(*								ELSIF iVisionScanModel=0 THEN
									(* found nothing, check if there is a part *)
									IF bRetryVision THEN
										sCurrentState.eStep := SP_RunStp103;
										bRetryVision := FALSE;
									ELSE
										sCurrentState.eStep := SP_RunStp120;
									END_IF
								ELSIF iVisionScanModel < iMaxScanVisionModelPart THEN
									(* relaunch scan with next step model *)
									iVisionScanModel := iVisionScanModel + 1;
									sCurrentState.eStep := SP_RunStp105;
								ELSE
									(* Part cannot be recognize, skip to next one *)
									aTPartOnPlate[LPP_Lift1,iPlatePos].ePartStatus := PPS_BadPart;
									iPlatePos := iPlatePos + 1;
									sCurrentState.eStep := SP_RunStp102;
*)								END_IF
							END_IF
						SP_RunStp110: (* Found valid position, Get Z position *)
							IF bUse103171OptimB3 THEN
								IF (alrZLiftPos[LTP_Lift1] = 0) THEN
									eScanPos := LTP_Lift1;
									eReturnStepMeasureZLift := SP_RunStp110;
									sCurrentState.eStep := SP_RunStp500;
								ELSE
									ZPositionTakeGive := alrRobotPos[LTA_Z,LTP_TableSideALayering1] + alrRobotOffset[LTA_Z, iHead] + (lrCalibrationPartAndHeadHeight - sPartDataMMI.lrPartAndHeadHeight) - alrZLiftPos[LTP_Lift1] - lrZSensorCalibrationOffset;
									sCurrentState.eStep := SP_RunStp114;
								END_IF
							ELSE
								iZSensorPositionScan := 0;
								sCurrentState.eStep := SP_RunStp111;
							END_IF
						SP_RunStp111:
							alrSecuredTarget[LA_X] := alrRobotPos[LTA_X,LTP_Lift1] + alrRobotOffset[LTA_X, LTO_ZSensor] + alrLiftCalibrationOffset[LTP_Lift1,LTA_X]  -  sPlateData.alrPartOnPlate[iPlatePos].lrX - sPartDataMMI.alrSensorZOffset[iZSensorPositionScan].lrX;
							alrSecuredTarget[LA_Y] :=alrRobotPos[LTA_Y,LTP_Lift1] + alrRobotOffset[LTA_Y, LTO_ZSensor] + alrLiftCalibrationOffset[LTP_Lift1,LTA_Y] - sPlateData.alrPartOnPlate[iPlatePos].lrY - sPartDataMMI.alrSensorZOffset[iZSensorPositionScan].lrY;
							TSensorZWaitStab(IN := FALSE);
							sCurrentState.bWaitStep := TRUE;
							eReturnStep4SecureMove := SP_RunStp112;
							sCurrentState.eStep := SP_RunStp550;
						SP_RunStp112:
							IF eRobotXYTStatus = AS_InPosition THEN
								TSensorZWaitStab(IN := TRUE, PT := TSensorZWaitStabTime);
								IF TSensorZWaitStab.Q THEN
									IF TSensorMeasure.bInputOutOfRange THEN
										bZSensorOutOfRangeError := TRUE;
									END_IF
									lrZSensorPosition[iZSensorPositionScan] := TSensorMeasure.lrValue;
									IF iZSensorPositionScan = 0 AND (sPartDataMMI.alrSensorZOffset[1].lrX<>0 OR sPartDataMMI.alrSensorZOffset[1].lrY<>0) THEN
										iZSensorPositionScan := iZSensorPositionScan + 1;
										sCurrentState.eStep := SP_RunStp111;
									ELSE
										sCurrentState.eStep := SP_RunStp113;
									END_IF
								END_IF
							END_IF
						SP_RunStp113:
							IF iZSensorPositionScan = 1 THEN
								(* We used two position, mean the value *)
								ZPositionTakeGive := (lrZSensorPosition[0] + lrZSensorPosition[1]) / 2;
							ELSE
								(* Only one position, use the first one then *)
								ZPositionTakeGive := lrZSensorPosition[0];
							END_IF
							ZPositionTakeGive := alrRobotPos[LTA_Z,LTP_TableSideALayering1] + alrRobotOffset[LTA_Z, iHead] + (lrCalibrationPartAndHeadHeight - sPartDataMMI.lrPartAndHeadHeight) - ZPositionTakeGive;
							sCurrentState.eStep := SP_RunStp114;
						SP_RunStp114: (* Move to take position *)
							IF sRunDataVision.TVisionPartData.bPresent AND NOT sRunDataVision.TVisionPartData.bValid THEN
								alrSecuredTarget[LA_X] := alrRobotPos[LTA_X,LTP_Lift1] + alrRobotOffset[LTA_X, iHead] + alrLiftCalibrationOffset[LTP_Lift1,LTA_X]  -  sPlateData.alrPartOnPlate[iPlatePos].lrX;	// + INT(iPlatePos/5) * 1/9 * offsetXMax;		// HFO : when vision diseable, correct the offset X between parts 
								alrSecuredTarget[LA_Y] :=alrRobotPos[LTA_Y,LTP_Lift1] + alrRobotOffset[LTA_Y, iHead] + alrLiftCalibrationOffset[LTP_Lift1,LTA_Y] - sPlateData.alrPartOnPlate[iPlatePos].lrY;	// + int(iPlatePos%5) * 1/4 * offsetYMax;		// HFO : when vision diseable, correct the offset Y between parts 
								alrTargetPos[LA_THETA] := alrRobotPos[LTA_THETA,LTP_TableSideALayering1] + alrRobotOffset[LTA_THETA, iHead] - (-90);
							ELSE
								alrSecuredTarget[LA_X] := alrRobotPos[LTA_X,LTP_Lift1] + alrRobotOffset[LTA_X, iHead] + alrLiftCalibrationOffset[LTP_Lift1,LTA_X]  -  sPlateData.alrPartOnPlate[iPlatePos].lrX + sRunDataVision.TVisionPartData.lrX;
								alrSecuredTarget[LA_Y] :=alrRobotPos[LTA_Y,LTP_Lift1] + alrRobotOffset[LTA_Y, iHead] + alrLiftCalibrationOffset[LTP_Lift1,LTA_Y] - sPlateData.alrPartOnPlate[iPlatePos].lrY + sRunDataVision.TVisionPartData.lrY;
								alrTargetPos[LA_THETA] := alrRobotPos[LTA_THETA,LTP_TableSideALayering1] + alrRobotOffset[LTA_THETA, iHead] + (360 - sRunDataVision.TVisionPartData.lrTheta);
							END_IF
							aeMoveRobotCommand[LA_THETA] := AC_MoveAtAbsPos;
							eReturnStep4SecureMove := SP_RunStp115;
							sCurrentState.eStep := SP_RunStp550;
						SP_RunStp115:
							IF eRobotXYTStatus = AS_InPosition THEN
								sCurrentState.eStep := SP_RunStp1;
							END_IF
						SP_RunStp120: (*Scan Vision Empty position *)
							sRunDataVision.iUseModel := iVisionModelEmpty;
							eVisionRunCmd := RCV_AnalyseImage;
							sCurrentState.eStep := SP_RunStp121;
						SP_RunStp121: (* Check for empty position *)
							IF eVisionRunStatus = RS_WaitRequest THEN
								IF NOT sRunDataVision.TVisionPartData.bPresent THEN
									(* Found Empty Position *)
									aTPartOnPlate[LPP_Lift1,iPlatePos].ePartStatus := PPS_Absent;
									iPlatePos := iPlatePos + 1;
									sCurrentState.eStep := SP_RunStp102;
								ELSE
									(*  Position is not empty, part is not recognize*)
									iVisionScanModel := iVisionScanModel + 1;
									sCurrentState.eStep := SP_RunStp104;
								END_IF
							END_IF
						SP_RunStp150: (* Switch plate *)
							bInvalidPlate := FALSE;
							FOR iPlatePos := 0 TO sPlateData.iNbPartOnPlate-1 DO
								IF aTPartOnPlate[LPP_Lift1,iPlatePos].ePartStatus = PPS_BadPart THEN
//									bInvalidPlate := TRUE;
									EXIT;
								END_IF
							END_FOR
							IF bInvalidPlate THEN
								(* goto invalid plate *)
								bLift1Lift1BadPlate := TRUE;
								eLift1RunCmd := RCL_MoveToOpenDrawer;
								sCurrentState.eStep := SP_RunStp101;
							ELSE
								sCurrentState.eStep := SP_RunStp70; (* Call Switch Plate *)
								eReturnStep := SP_RunStp101;
							END_IF
						SP_RunStp170: (*Get from Table *)
							IF eTableSide = TS_A THEN
								IF sRunData.iLayringPos = 0 THEN
									ePos := LTP_TableSideALayering1;
								ELSE
									ePos := LTP_TableSideALayering2;
								END_IF
							ELSE
								IF sRunData.iLayringPos = 0 THEN
									ePos := LTP_TableSideBLayering1;
								ELSE
									ePos := LTP_TableSideBLayering2;
								END_IF
							END_IF
							alrSecuredTarget[LA_X] := alrRobotPos[LTA_X,ePos] + alrRobotOffset[LTA_X, iHead];
							alrSecuredTarget[LA_Y] :=  alrRobotPos[LTA_Y,ePos] + alrRobotOffset[LTA_Y, iHead];
							alrTargetPos[LA_THETA] := alrRobotPos[LTA_THETA,ePos] + alrRobotOffset[LTA_THETA, iHead];
							ZPositionTakeGive := alrRobotPos[LTA_Z,ePos] + alrRobotOffset[LTA_Z, iHead];
							alrSecuredTarget[LA_X] := alrSecuredTarget[LA_X]   -  sPartDataMMI.alrPartOffsetLayering[sRunData.iLayringOffsetPos].lrX;
							alrSecuredTarget[LA_Y] := alrSecuredTarget[LA_Y]  + sPartDataMMI.alrPartOffsetLayering[sRunData.iLayringOffsetPos].lrY;
							ZPositionTakeGive := ZPositionTakeGive + (lrCalibrationLayeringAndPartAndHeadHeight - sPartDataMMI.lrLayeringAndPartAndHeadHeight);
							aeMoveRobotCommand[LA_THETA] := AC_MoveAtAbsPos;
							eReturnStep4SecureMove := SP_RunStp171;
							sCurrentState.eStep := SP_RunStp550;
						SP_RunStp171:
							IF eRobotXYTStatus = AS_InPosition THEN
								sCurrentState.eStep := SP_RunStp1;
							END_IF
						SP_RunStp180: (*Get from Turn Over *)
							alrSecuredTarget[LA_X] := alrRobotPos[LTA_X,LTP_TurnOverFix] + alrRobotOffset[LTA_X, iHead];
							alrSecuredTarget[LA_Y] :=  alrRobotPos[LTA_Y,LTP_TurnOverFix] + alrRobotOffset[LTA_Y, iHead];
							alrTargetPos[LA_THETA] := alrRobotPos[LTA_THETA,LTP_TurnOverFix] + alrRobotOffset[LTA_THETA, iHead];
							ZPositionTakeGive := alrRobotPos[LTA_Z,LTP_TurnOverFix] + alrRobotOffset[LTA_Z, iHead];
							ZPositionTakeGive := ZPositionTakeGive +  (lrCalibrationLayeringAndPartAndHeadHeight - sPartDataMMI.lrLayeringAndPartAndHeadHeight);
							aeMoveRobotCommand[LA_THETA] := AC_MoveAtAbsPos;
							eReturnStep4SecureMove := SP_RunStp181;
							sCurrentState.eStep := SP_RunStp550;
						SP_RunStp181:
							IF eRobotXYTStatus = AS_InPosition THEN
								sCurrentState.eStep := SP_RunStp1;
							END_IF
						SP_RunStp200 : (*Prepare for Drop part*)
							CASE sRunData.eModule OF
								LMP_Reject, LMP_Sample:
									sCurrentState.eStep := SP_RunStp301;
								LMP_Lift2:
									IF sPartDataMMI.bDropInBox THEN
										sCurrentState.eStep := SP_RunStp230;
									ELSE
										sCurrentState.eStep := SP_RunStp201;
									END_IF
								LMP_Table:
									sCurrentState.eStep := SP_RunStp270;
								LMP_TurnOverArm:
									sCurrentState.eStep := SP_RunStp280;
							END_CASE
						SP_RunStp201: (* Check Lift Status*)
							IF eLift2RunStatus = RS_WaitRequest THEN
								CASE sLift2RunData.eLiftPos OF
									LP_OnPlate:
										iPlatePos := 0;
										sCurrentState.eStep := SP_RunStp202;
									LP_Full,LP_Empty:
										bLift2NeedsPlate := TRUE;
										eLift2RunCmd := RCL_MoveToOpenDrawer;
								ELSE
									eLift2RunCmd := RCL_MoveToPlate;
								END_CASE
							END_IF
						SP_RunStp202: (*Check part status*)
							bFoundPlatePos := FALSE;
							WHILE (iPlatePos < sPlateData.iNbPartOnPlate) DO
								IF aTPartOnPlate[LPP_Lift2,iPlatePos].ePartStatus = PPS_Absent OR aTPartOnPlate[LPP_Lift2,iPlatePos].ePartStatus = PPS_Undefined THEN
									bFoundPlatePos := TRUE;
									EXIT;
								ELSE
									iPlatePos := iPlatePos + 1;
								END_IF
							END_WHILE
							IF NOT bFoundPlatePos THEN
								(* Goto switch plate *)
								sCurrentState.eStep := SP_RunStp250;
							ELSE
								IF aTPartOnPlate[LPP_Lift2,iPlatePos].ePartStatus = PPS_Absent OR (NOT sPlateData.bUseVisionForDrop OR bDisableVision) THEN
									sCurrentState.eStep := SP_RunStp210;
								ELSE
									sCurrentState.eStep := SP_RunStp203;
								END_IF
							END_IF
						SP_RunStp203: (*Scan Vision Part Position *)
							alrSecuredTarget[LA_X] := alrRobotPos[LTA_X,LTP_Lift2] + alrRobotOffset[LTA_X, LTO_Vision] + alrLiftCalibrationOffset[LTP_Lift2,LTA_X]  - sPlateData.alrPartOnPlate[iPlatePos].lrX ;
							alrSecuredTarget[LA_Y] :=  alrRobotPos[LTA_Y,LTP_Lift2] + alrRobotOffset[LTA_Y, LTO_Vision] + alrLiftCalibrationOffset[LTP_Lift2,LTA_Y] - sPlateData.alrPartOnPlate[iPlatePos].lrY ;
							iVisionScanModel := 0;
							TVisionWaitStab(IN := FALSE);
							eReturnStep4SecureMove := SP_RunStp204;
							sCurrentState.eStep := SP_RunStp550;
						SP_RunStp204:
							IF eRobotXYTStatus = AS_InPosition THEN
								IF aTPartOnPlate[LPP_Lift2,iPlatePos].ePartStatus = PPS_Absent THEN
									sCurrentState.eStep := SP_RunStp208;
								ELSE
									TVisionWaitStab(IN := TRUE, PT := TVisionWaitStabTime);
									IF TVisionWaitStab.Q THEN
										eVisionRunCmd := RCV_GrabImage;
										sCurrentState.eStep := SP_RunStp205;
									END_IF
								END_IF
							END_IF
						SP_RunStp205: (* Move to pre-drop position *)
							IF eVisionRunStatus = RS_WaitRequest THEN
								IF bUse103171OptimB5PreMoveXY THEN
									alrSecuredTarget[LA_X] := alrRobotPos[LTA_X,LTP_Lift2] + alrRobotOffset[LTA_X, iHead] + alrLiftCalibrationOffset[LTP_Lift2,LTA_X]  -  sPlateData.alrPartOnPlate[iPlatePos].lrX;
									alrSecuredTarget[LA_Y] :=alrRobotPos[LTA_Y,LTP_Lift2] + alrRobotOffset[LTA_Y, iHead] + alrLiftCalibrationOffset[LTP_Lift2,LTA_Y] - sPlateData.alrPartOnPlate[iPlatePos].lrY;
									alrTargetPos[LA_THETA] := alrRobotPos[LTA_THETA,LTP_TableSideALayering1] + alrRobotOffset[LTA_THETA, iHead];
									aeMoveRobotCommand[LA_THETA] := AC_MoveAtAbsPos;
									eReturnStep4SecureMove := SP_RunStp207;
									sCurrentState.eStep := SP_RunStp550;
								ELSE
									sCurrentState.eStep := SP_RunStp207;
								END_IF
								sRunDataVision.iUseModel := iVisionModelEmpty;
								eVisionRunCmd := RCV_AnalyseImage;
							END_IF
						SP_RunStp207: (* Check for part *)
							IF eVisionRunStatus = RS_WaitRequest THEN
								IF NOT sRunDataVision.TVisionPartData.bPresent THEN
									(* Found empty position *)
									aTPartOnPlate[LPP_Lift2,iPlatePos].ePartStatus := PPS_Absent;
									sCurrentState.eStep := SP_RunStp208;
								ELSE
									(* found something *)
									aTPartOnPlate[LPP_Lift2,iPlatePos].ePartStatus := PPS_Present;
									iPlatePos := iPlatePos + 1;
									sCurrentState.eStep := SP_RunStp202;
								END_IF
							END_IF
						SP_RunStp208: (*Scan Vision for position *)
							IF sPlateData.bUseVisionForDrop THEN
								sRunDataVision.iUseModel := aiVisionModelPlate[iVisionScanModel];
								eVisionRunCmd := RCV_AnalyseImage;
								sCurrentState.eStep := SP_RunStp209;
							ELSE
								sCurrentState.eStep := SP_RunStp210;
							END_IF
						SP_RunStp209: (* Get position *)
							IF eVisionRunStatus = RS_WaitRequest THEN
								IF (*sRunDataVision.TVisionPartData.bPresent AND*) sRunDataVision.TVisionPartData.bValid THEN
									(* Found valide position *)
									sCurrentState.eStep := SP_RunStp210;
								(*ELSIF sRunDataVision.TVisionPartData.bPresent AND NOT sRunDataVision.TVisionPartData.bValid THEN
									(* Found invalide part, relaunch with other model ??? not implemented right now*)
									aTPartOnPlate[LPP_Lift2,iPlatePos].ePartStatus := PPS_BadPart;
									iPlatePos := iPlatePos + 1;
									sCurrentState.eStep := SP_RunStp202;*)
								ELSIF iVisionScanModel < iMaxScanVisionModelPlate THEN
									(* relaunch scan with next step model *)
									iVisionScanModel := iVisionScanModel + 1;
									sCurrentState.eStep := SP_RunStp208;
								ELSE
									(* Plate cannot be recognize, skip to next one *)
									aTPartOnPlate[LPP_Lift2,iPlatePos].ePartStatus := PPS_BadPart;
									iPlatePos := iPlatePos + 1;
									sCurrentState.eStep := SP_RunStp202;
								END_IF
							END_IF
						SP_RunStp210: (* Found valid position, Get Z position *)
							IF bUse103171OptimB3 THEN
								IF (alrZLiftPos[LTP_Lift2] = 0) THEN
									eScanPos := LTP_Lift2;
									eReturnStepMeasureZLift := SP_RunStp210;
									sCurrentState.eStep := SP_RunStp500;
								ELSE
									ZPositionTakeGive := alrRobotPos[LTA_Z,LTP_TableSideALayering1] + alrRobotOffset[LTA_Z, iHead] + (lrCalibrationPartAndHeadHeight - sPartDataMMI.lrPartAndHeadHeight) - alrZLiftPos[LTP_Lift2] - lrZSensorCalibrationOffset;
									//ZPositionTakeGive := alrRobotPos[LTA_Z,sRunData.eModule] + alrRobotOffset[LTA_Z, iHead] + (lrCalibrationPartAndHeadHeight - sPartDataMMI.lrPartAndHeadHeight) - alrZLiftPos[LTP_Lift2];
									sCurrentState.eStep := SP_RunStp214;
								END_IF
							ELSE
								iZSensorPositionScan := 0;
								sCurrentState.eStep := SP_RunStp211;
							END_IF
						SP_RunStp211: (* Calcul de la position x et y de mesure hauteur *)
							alrSecuredTarget[LA_X] := alrRobotPos[LTA_X,LTP_Lift2] + alrRobotOffset[LTA_X, LTO_ZSensor] + alrLiftCalibrationOffset[LTP_Lift2,LTA_X]  -  sPlateData.alrPartOnPlate[iPlatePos].lrX - sPartDataMMI.alrSensorZOffset[iZSensorPositionScan].lrX;
							alrSecuredTarget[LA_Y] :=alrRobotPos[LTA_Y,LTP_Lift2] + alrRobotOffset[LTA_Y, LTO_ZSensor] + alrLiftCalibrationOffset[LTP_Lift2,LTA_Y] - sPlateData.alrPartOnPlate[iPlatePos].lrY - sPartDataMMI.alrSensorZOffset[iZSensorPositionScan].lrY;
							TSensorZWaitStab(IN := FALSE);
							eReturnStep4SecureMove := SP_RunStp212;
							sCurrentState.eStep := SP_RunStp550;
						SP_RunStp212:
							IF eRobotXYTStatus = AS_InPosition THEN
								TSensorZWaitStab(IN := TRUE, PT := TSensorZWaitStabTime);
								IF TSensorZWaitStab.Q THEN
									IF TSensorMeasure.bInputOutOfRange THEN
										bZSensorOutOfRangeError := TRUE;
									END_IF
									lrZSensorPosition[iZSensorPositionScan] := TSensorMeasure.lrValue;
									IF iZSensorPositionScan = 0 AND (sPartDataMMI.alrSensorZOffset[1].lrX<>0 OR sPartDataMMI.alrSensorZOffset[1].lrY<>0) THEN
										iZSensorPositionScan := iZSensorPositionScan + 1;
										sCurrentState.eStep := SP_RunStp211;
									ELSE
										sCurrentState.eStep := SP_RunStp213;
									END_IF
								END_IF
							END_IF
						SP_RunStp213:
							IF iZSensorPositionScan = 1 THEN
								(* We used two position, mean the value *)
								ZPositionTakeGive := (lrZSensorPosition[0] + lrZSensorPosition[1]) / 2;
							ELSE
								(* Only one position, use the first one then *)
								ZPositionTakeGive := lrZSensorPosition[0];
							END_IF
							ZPositionTakeGive := alrRobotPos[LTA_Z,LTP_TableSideALayering1] + alrRobotOffset[LTA_Z, iHead] + (lrCalibrationPartAndHeadHeight - sPartDataMMI.lrPartAndHeadHeight) - ZPositionTakeGive;
							sCurrentState.eStep := SP_RunStp214;
						SP_RunStp214: (* Move to take position *)
							alrSecuredTarget[LA_X] := alrRobotPos[LTA_X,LTP_Lift2] + alrRobotOffset[LTA_X, iHead] + alrLiftCalibrationOffset[LTP_Lift2,LTA_X]  -  sPlateData.alrPartOnPlate[iPlatePos].lrX;
							alrSecuredTarget[LA_Y] := alrRobotPos[LTA_Y,LTP_Lift2] + alrRobotOffset[LTA_Y, iHead] + alrLiftCalibrationOffset[LTP_Lift2,LTA_Y] - sPlateData.alrPartOnPlate[iPlatePos].lrY;
							alrTargetPos[LA_THETA] := alrRobotPos[LTA_THETA,LTP_TableSideALayering1] + alrRobotOffset[LTA_THETA, iHead];
							IF sPlateData.bUseVisionForDrop THEN
								TComputeVisionPos( THead := sPartDataMMI.THeadOffset, lrAngle := sRunDataVision.TVisionPartData.lrTheta, TOffsetPos => TOffsetPos);
								alrSecuredTarget[LA_X] := alrSecuredTarget[LA_X] + sRunDataVision.TVisionPartData.lrX - TOffsetPos.lrX;
								alrSecuredTarget[LA_Y] := alrSecuredTarget[LA_Y] + sRunDataVision.TVisionPartData.lrY + TOffsetPos.lrY;
								alrTargetPos[LA_THETA] := alrTargetPos[LA_THETA] + TOffsetPos.lrTheta;
							ELSE
								alrTargetPos[LA_THETA] := alrTargetPos[LA_THETA] + sPartDataMMI.lrPartOffsetThetaLiftDrop;	// + lrThetaOffsetMecDrop;		// var ajoutée en comparaison avec la vision
								alrSecuredTarget[LA_X] := alrSecuredTarget[LA_X] + sPartDataMMI.lrPartOffsetXLiftDrop;		// + lrXOffsetMecDrop;					// valueur ajoutée en comparaison avec la vision
								alrSecuredTarget[LA_Y] := alrSecuredTarget[LA_Y] + sPartDataMMI.lrPartOffsetYLiftDrop;		// + lrYOffsetMecDrop;
							END_IF
							aeMoveRobotCommand[LA_THETA] := AC_MoveAtAbsPos;
							eReturnStep4SecureMove := SP_RunStp215;
							sCurrentState.eStep := SP_RunStp550;
						SP_RunStp215:
							IF eRobotXYTStatus = AS_InPosition THEN
								sCurrentState.eStep := SP_RunStp1;
							END_IF
						SP_RunStp230:
							alrSecuredTarget[LA_X] := alrRobotPos[LTA_X,LTP_BulkBox] + alrRobotOffset[LTA_X, iHead];
							alrSecuredTarget[LA_Y] :=alrRobotPos[LTA_Y,LTP_BulkBox] + alrRobotOffset[LTA_Y, iHead];
							alrTargetPos[LA_THETA] := alrRobotPos[LTA_THETA,LTP_TableSideALayering1] + alrRobotOffset[LTA_THETA, iHead];
							aeMoveRobotCommand[LA_THETA] := AC_MoveAtAbsPos;
							eReturnStep4SecureMove := SP_RunStp231;
							sCurrentState.eStep := SP_RunStp550;
						SP_RunStp231:
							IF eRobotXYTStatus = AS_InPosition THEN
								sCurrentState.eStep := SP_RunStp1;
							END_IF
						SP_RunStp250: (* Switch plate *)
							bPlateEmpty := TRUE;
							FOR iPlatePos := 0 TO sPlateData.iNbPartOnPlate-1 DO
								IF aTPartOnPlate[LPP_Lift1,iPlatePos].ePartStatus <> PPS_Absent THEN
									bPlateEmpty := FALSE;
									EXIT;
								END_IF
							END_FOR
							IF bPlateEmpty THEN
								sCurrentState.eStep := SP_RunStp70; (* Call Switch Plate *)
								eReturnStep := SP_RunStp201;
							ELSE
								bDoPlateScan := TRUE;
								FOR iPlatePos := 0 TO sPlateData.iNbPartOnPlate-1 DO
									IF aTPartOnPlate[LPP_Lift1,iPlatePos].ePartStatus <> PPS_Undefined AND aTPartOnPlate[LPP_Lift1,iPlatePos].ePartStatus <> PPS_Absent THEN
										bDoPlateScan := FALSE;
										EXIT;
									END_IF
								END_FOR
								IF bDoPlateScan THEN
									sCurrentState.eStep := SP_RunStp251;
								ELSE
									(* goto invalid plate *)
									bLift2NeedsPlate := TRUE;
									eLift2RunCmd := RCL_MoveToOpenDrawer;
									sCurrentState.eStep := SP_RunStp201;
								END_IF
							END_IF
						SP_RunStp251: (*Find first undefined pos *)
							bFoundPlatePos := FALSE;
							iPlatePos := 0;
							WHILE (iPlatePos < sPlateData.iNbPartOnPlate) DO
								IF aTPartOnPlate[LPP_Lift1,iPlatePos].ePartStatus = PPS_Undefined THEN
									bFoundPlatePos := TRUE;
									EXIT;
								ELSE
									iPlatePos := iPlatePos + 1;
								END_IF
							END_WHILE
							IF NOT bFoundPlatePos THEN
								(* goto invalid plate *)
								bLift2NeedsPlate := TRUE;
								eLift2RunCmd := RCL_MoveToOpenDrawer;
								sCurrentState.eStep := SP_RunStp201;
							ELSE
								sCurrentState.eStep := SP_RunStp252;
							END_IF
						SP_RunStp252: (*Scan Vision Part Position *)
							alrSecuredTarget[LA_X] := alrRobotPos[LTA_X,LTP_Lift1] + alrRobotOffset[LTA_X, LTO_Vision] + alrLiftCalibrationOffset[LTP_Lift1,LTA_X]  - sPlateData.alrPartOnPlate[iPlatePos].lrX ;
							alrSecuredTarget[LA_Y] :=  alrRobotPos[LTA_Y,LTP_Lift1] + alrRobotOffset[LTA_Y, LTO_Vision] + alrLiftCalibrationOffset[LTP_Lift1,LTA_Y] - sPlateData.alrPartOnPlate[iPlatePos].lrY ;
							TVisionWaitStab(IN := FALSE);
							eReturnStep4SecureMove := SP_RunStp253;
							sCurrentState.eStep := SP_RunStp550;
						SP_RunStp253:
							IF eRobotXYTStatus = AS_InPosition THEN
								TVisionWaitStab(IN := TRUE, PT := TVisionWaitStabTime);
								IF TVisionWaitStab.Q THEN
									eVisionRunCmd := RCV_GrabImage;
									sCurrentState.eStep := SP_RunStp254;
								END_IF
							END_IF
						SP_RunStp254:
							IF eVisionRunStatus = RS_WaitRequest THEN
								sRunDataVision.iUseModel := iVisionModelEmpty;
								eVisionRunCmd := RCV_AnalyseImage;
								sCurrentState.eStep := SP_RunStp255;
							END_IF
						SP_RunStp255: (* Check for part *)
							IF eVisionRunStatus = RS_WaitRequest THEN
								IF NOT sRunDataVision.TVisionPartData.bPresent THEN
									(* Found empty position *)
									aTPartOnPlate[LPP_Lift1,iPlatePos].ePartStatus := PPS_Absent;
									iPlatePos := iPlatePos + 1;
									IF (iPlatePos < sPlateData.iNbPartOnPlate) THEN
										sCurrentState.eStep := SP_RunStp252;
									ELSE
										(* All position on lift1 plate is empty, we can switch plate then *)
										sCurrentState.eStep := SP_RunStp70; (* Call Switch Plate *)
										eReturnStep := SP_RunStp201;
									END_IF
								ELSE
									(* goto invalid plate *)
									bLift2NeedsPlate := TRUE;
									eLift2RunCmd := RCL_MoveToOpenDrawer;
									sCurrentState.eStep := SP_RunStp201;
								END_IF
							END_IF
						SP_RunStp270: (*Give to Table *)
							IF eTableSide = TS_A THEN
								IF sRunData.iLayringPos = 0 THEN
									ePos := LTP_TableSideALayering1;
								ELSE
									ePos := LTP_TableSideALayering2;
								END_IF
							ELSE
								IF sRunData.iLayringPos = 0 THEN
									ePos := LTP_TableSideBLayering1;
								ELSE
									ePos := LTP_TableSideBLayering2;
								END_IF
							END_IF
							alrSecuredTarget[LA_X] := alrRobotPos[LTA_X,ePos] + alrRobotOffset[LTA_X, iHead];
							alrSecuredTarget[LA_Y] := alrRobotPos[LTA_Y,ePos] + alrRobotOffset[LTA_Y, iHead];
							alrTargetPos[LA_THETA] := alrRobotPos[LTA_THETA,ePos] + alrRobotOffset[LTA_THETA, iHead];
							ZPositionTakeGive := alrRobotPos[LTA_Z,ePos] + alrRobotOffset[LTA_Z, iHead];
							alrSecuredTarget[LA_X] := alrSecuredTarget[LA_X] - sPartDataMMI.alrPartOffsetLayering[sRunData.iLayringOffsetPos].lrX;
							alrSecuredTarget[LA_Y] := alrSecuredTarget[LA_Y] + sPartDataMMI.alrPartOffsetLayering[sRunData.iLayringOffsetPos].lrY;
							ZPositionTakeGive := ZPositionTakeGive + (lrCalibrationLayeringAndPartAndHeadHeight - sPartDataMMI.lrLayeringAndPartAndHeadHeight);
							aeMoveRobotCommand[LA_THETA] := AC_MoveAtAbsPos;
							eReturnStep4SecureMove := SP_RunStp271;
							sCurrentState.eStep := SP_RunStp550;
						SP_RunStp271:
							IF eRobotXYTStatus = AS_InPosition THEN
								sCurrentState.eStep := SP_RunStp1;
							END_IF
						SP_RunStp280: (*Get from Turn Over *)
							alrSecuredTarget[LA_X] := alrRobotPos[LTA_X,LTP_TurnOverArm] + alrRobotOffset[LTA_X, iHead];
							alrSecuredTarget[LA_Y] :=  alrRobotPos[LTA_Y,LTP_TurnOverArm] + alrRobotOffset[LTA_Y, iHead];
							alrTargetPos[LA_THETA] := alrRobotPos[LTA_THETA,LTP_TurnOverArm] + alrRobotOffset[LTA_THETA, iHead];
							ZPositionTakeGive := alrRobotPos[LTA_Z,LTP_TurnOverArm] + alrRobotOffset[LTA_Z, iHead];
							ZPositionTakeGive := ZPositionTakeGive + (lrCalibrationHeadSusPartHeadSousHeight - sPartDataMMI.lrHeadSusPartHeadSousHeight);
							aeMoveRobotCommand[LA_THETA] := AC_MoveAtAbsPos;
							eReturnStep4SecureMove := SP_RunStp281;
							sCurrentState.eStep := SP_RunStp550;
						SP_RunStp281:
							IF eRobotXYTStatus = AS_InPosition THEN
								sCurrentState.eStep := SP_RunStp1;
							END_IF
						SP_RunStp301: (* Check Reject Status*)
							IF eRejectRunStatus = RS_WaitRequest THEN
								CASE sRejectRunData.eRejectStatus OF
									RS_Ready:
										eRejectRunCmd := RCR_LockDrawer;
									RS_Locked:
										IF sRunData.eModule = LMP_Sample THEN
											iPlatePos := sPlateData.iNbPartOnPlate - 1;
										ELSE
											iPlatePos := 0;
										END_IF
										sCurrentState.eStep := SP_RunStp302;
										IF sPartDataMMI.bDropInBox THEN
											sCurrentState.eStep := SP_RunStp330;
										END_IF
									ELSE
										bRejectNeedsPlate := TRUE;
										eRejectRunCmd := RCR_OpenDrawer;
								END_CASE
							END_IF
						SP_RunStp302: (*Check part status*)
							bFoundPlatePos := FALSE;
							IF sRunData.eModule = LMP_Sample THEN
								WHILE (iPlatePos >= 0) DO
									IF aTPartOnPlate[LPP_Reject,iPlatePos].ePartStatus = PPS_Absent OR aTPartOnPlate[LPP_Reject,iPlatePos].ePartStatus = PPS_Undefined THEN
										bFoundPlatePos := TRUE;
										EXIT;
									ELSE
										iPlatePos := iPlatePos - 1;
									END_IF
								END_WHILE
							ELSE
								WHILE (iPlatePos < sPlateData.iNbPartOnPlate) DO
									IF aTPartOnPlate[LPP_Reject,iPlatePos].ePartStatus = PPS_Absent OR aTPartOnPlate[LPP_Reject,iPlatePos].ePartStatus = PPS_Undefined THEN
										bFoundPlatePos := TRUE;
										EXIT;
									ELSE
										iPlatePos := iPlatePos + 1;
									END_IF
								END_WHILE
							END_IF
							IF NOT bFoundPlatePos THEN
								(* Request new plate *)
								bRejectNeedsPlate := TRUE;
								eRejectRunCmd := RCR_OpenDrawer;
								sCurrentState.eStep := SP_RunStp301;
							ELSE
								IF bDisableVision OR NOT sPlateData.bUseVisionForDrop THEN
									sCurrentState.eStep := SP_RunStp310;
								ELSE
									sCurrentState.eStep := SP_RunStp303;
								END_IF
							END_IF
						SP_RunStp303: (*Scan Vision Part Position *)
							alrSecuredTarget[LA_X] := alrRobotPos[LTA_X,LTP_Reject] + alrRobotOffset[LTA_X, LTO_Vision] + alrLiftCalibrationOffset[LTP_Reject,LTA_X]  - sPlateData.alrPartOnPlate[iPlatePos].lrX ;
							alrSecuredTarget[LA_Y] :=  alrRobotPos[LTA_Y,LTP_Reject] + alrRobotOffset[LTA_Y, LTO_Vision] + alrLiftCalibrationOffset[LTP_Reject,LTA_Y] - sPlateData.alrPartOnPlate[iPlatePos].lrY ;
							iVisionScanModel := 0;
							TVisionWaitStab(IN := FALSE);
							eReturnStep4SecureMove := SP_RunStp304;
							sCurrentState.eStep := SP_RunStp550;
						SP_RunStp304:
							IF eRobotXYTStatus = AS_InPosition THEN
								TVisionWaitStab(IN := TRUE, PT := TVisionWaitStabTime);
								IF TVisionWaitStab.Q THEN
									eVisionRunCmd := RCV_GrabImage;
									sCurrentState.eStep := SP_RunStp305;
								END_IF
							END_IF
						SP_RunStp305: (* Move to pre-drop position *)
							IF eVisionRunStatus = RS_WaitRequest THEN
								IF bUse103171OptimB5PreMoveXY THEN
									alrSecuredTarget[LA_X] := alrRobotPos[LTA_X,LTP_Reject] + alrRobotOffset[LTA_X, iHead] + alrLiftCalibrationOffset[LTP_Reject,LTA_X]  -  sPlateData.alrPartOnPlate[iPlatePos].lrX;
									alrSecuredTarget[LA_Y] :=alrRobotPos[LTA_Y,LTP_Reject] + alrRobotOffset[LTA_Y, iHead] + alrLiftCalibrationOffset[LTP_Reject,LTA_Y] - sPlateData.alrPartOnPlate[iPlatePos].lrY;
									alrTargetPos[LA_THETA] := alrRobotPos[LTA_THETA,LTP_TableSideALayering1] + alrRobotOffset[LTA_THETA, iHead];
									aeMoveRobotCommand[LA_THETA] := AC_MoveAtAbsPos;
									eReturnStep4SecureMove := SP_RunStp307;
									sCurrentState.eStep := SP_RunStp550;
								ELSE
									sCurrentState.eStep := SP_RunStp307;
								END_IF
								sRunDataVision.iUseModel := iVisionModelEmpty;
								eVisionRunCmd := RCV_AnalyseImage;
							END_IF
						SP_RunStp307: (* Check for part *)
							IF eVisionRunStatus = RS_WaitRequest THEN
								IF NOT sRunDataVision.TVisionPartData.bPresent THEN
									(* Found empty position *)
									aTPartOnPlate[LPP_Reject,iPlatePos].ePartStatus := PPS_Absent;
									sCurrentState.eStep := SP_RunStp308;
								ELSE
									(* found something *)
									aTPartOnPlate[LPP_Reject,iPlatePos].ePartStatus := PPS_Present;
									IF sRunData.eModule = LMP_Sample THEN
										iPlatePos := iPlatePos - 1;
									ELSE
										iPlatePos := iPlatePos + 1;
									END_IF
									sCurrentState.eStep := SP_RunStp302;
								END_IF
							END_IF
						SP_RunStp308: (*Scan Vision for position *)
							IF sPlateData.bUseVisionForDrop THEN
								sRunDataVision.iUseModel := aiVisionModelPlate[iVisionScanModel];
								eVisionRunCmd := RCV_AnalyseImage;
								sCurrentState.eStep := SP_RunStp309;
							ELSE
								sCurrentState.eStep := SP_RunStp310;
							END_IF
						SP_RunStp309: (* Get position *)
							IF eVisionRunStatus = RS_WaitRequest THEN
								IF (*sRunDataVision.TVisionPartData.bPresent AND*) sRunDataVision.TVisionPartData.bValid THEN
									(* Found valide position *)
									sCurrentState.eStep := SP_RunStp310;
								(*ELSIF sRunDataVision.TVisionPartData.bPresent AND NOT sRunDataVision.TVisionPartData.bValid THEN
									(* Found invalide part, relaunch with other model ??? not implemented right now*)
									aTPartOnPlate[LPP_Reject,iPlatePos].ePartStatus := PPS_BadPart;
									IF sRunData.eModule = LMP_Sample THEN
										iPlatePos := iPlatePos - 1;
									ELSE
										iPlatePos := iPlatePos + 1;
									END_IF
									sCurrentState.eStep := SP_RunStp302;*)
								ELSIF iVisionScanModel < iMaxScanVisionModelPlate THEN
									(* relaunch scan with next step model *)
									iVisionScanModel := iVisionScanModel + 1;
									sCurrentState.eStep := SP_RunStp308;
								ELSE
									(* Plate cannot be recognize, skip to next one *)
									aTPartOnPlate[LPP_Reject,iPlatePos].ePartStatus := PPS_BadPart;
									IF sRunData.eModule = LMP_Sample THEN
										iPlatePos := iPlatePos - 1;
									ELSE
										iPlatePos := iPlatePos + 1;
									END_IF
									sCurrentState.eStep := SP_RunStp302;
								END_IF
							END_IF
						SP_RunStp310: (* Found valid position, Get Z position *)
							IF bUse103171OptimB3 THEN
								IF (alrZLiftPos[LTP_Reject] = 0) THEN
									eScanPos := LTP_Reject;
									eReturnStepMeasureZLift := SP_RunStp310;
									sCurrentState.eStep := SP_RunStp500;
								ELSE
									ZPositionTakeGive := alrRobotPos[LTA_Z,LTP_TableSideALayering1] + alrRobotOffset[LTA_Z, iHead] + (lrCalibrationPartAndHeadHeight - sPartDataMMI.lrPartAndHeadHeight) - alrZLiftPos[LTP_Reject];
									sCurrentState.eStep := SP_RunStp314;
								END_IF
							ELSE
								iZSensorPositionScan := 0;
								sCurrentState.eStep := SP_RunStp311;
							END_IF
						SP_RunStp311:
							alrSecuredTarget[LA_X] := alrRobotPos[LTA_X,LTP_Reject] + alrRobotOffset[LTA_X, LTO_ZSensor] + alrLiftCalibrationOffset[LTP_Reject,LTA_X]  -  sPlateData.alrPartOnPlate[iPlatePos].lrX - sPartDataMMI.alrSensorZOffset[iZSensorPositionScan].lrX;
							alrSecuredTarget[LA_Y] :=alrRobotPos[LTA_Y,LTP_Reject] + alrRobotOffset[LTA_Y, LTO_ZSensor] + alrLiftCalibrationOffset[LTP_Reject,LTA_Y] - sPlateData.alrPartOnPlate[iPlatePos].lrY - sPartDataMMI.alrSensorZOffset[iZSensorPositionScan].lrY;
							TSensorZWaitStab(IN := FALSE);
							eReturnStep4SecureMove := SP_RunStp312;
							sCurrentState.eStep := SP_RunStp550;
						SP_RunStp312:
							IF eRobotXYTStatus = AS_InPosition THEN
								TSensorZWaitStab(IN := TRUE, PT := TSensorZWaitStabTime);
								IF TSensorZWaitStab.Q THEN
									IF TSensorMeasure.bInputOutOfRange THEN
										bZSensorOutOfRangeError := TRUE;
									END_IF
									lrZSensorPosition[iZSensorPositionScan] := TSensorMeasure.lrValue;
									IF iZSensorPositionScan = 0 AND (sPartDataMMI.alrSensorZOffset[1].lrX<>0 OR sPartDataMMI.alrSensorZOffset[1].lrY<>0) THEN
										iZSensorPositionScan := iZSensorPositionScan + 1;
										sCurrentState.eStep := SP_RunStp311;
									ELSE
										sCurrentState.eStep := SP_RunStp313;
									END_IF
								END_IF
							END_IF
						SP_RunStp313:
							IF iZSensorPositionScan = 1 THEN
								(* We used two position, mean the value *)
								ZPositionTakeGive := (lrZSensorPosition[0] + lrZSensorPosition[1]) / 2;
							ELSE
								(* Only one position, use the first one then *)
								ZPositionTakeGive := lrZSensorPosition[0];
							END_IF
							ZPositionTakeGive := alrRobotPos[LTA_Z,LTP_TableSideALayering1] + alrRobotOffset[LTA_Z, iHead] + (lrCalibrationPartAndHeadHeight - sPartDataMMI.lrPartAndHeadHeight) - ZPositionTakeGive;
							sCurrentState.eStep := SP_RunStp314;
						SP_RunStp314: (* Move to take position *)
							alrSecuredTarget[LA_X] := alrRobotPos[LTA_X,LTP_Reject] + alrRobotOffset[LTA_X, iHead] + alrLiftCalibrationOffset[LTP_Reject,LTA_X]  -  sPlateData.alrPartOnPlate[iPlatePos].lrX;
							alrSecuredTarget[LA_Y] :=alrRobotPos[LTA_Y,LTP_Reject] + alrRobotOffset[LTA_Y, iHead] + alrLiftCalibrationOffset[LTP_Reject,LTA_Y] - sPlateData.alrPartOnPlate[iPlatePos].lrY;
							alrTargetPos[LA_THETA] := alrRobotPos[LTA_THETA,LTP_TableSideALayering1] + alrRobotOffset[LTA_THETA, iHead];
							IF sPlateData.bUseVisionForDrop THEN
								TComputeVisionPos( THead := sPartDataMMI.THeadOffset, lrAngle := sRunDataVision.TVisionPartData.lrTheta, TOffsetPos => TOffsetPos);
								alrSecuredTarget[LA_X] := alrSecuredTarget[LA_X] + sRunDataVision.TVisionPartData.lrX - TOffsetPos.lrX;
								alrSecuredTarget[LA_Y] := alrSecuredTarget[LA_Y] + sRunDataVision.TVisionPartData.lrY + TOffsetPos.lrY;
								alrTargetPos[LA_THETA] := alrTargetPos[LA_THETA] + TOffsetPos.lrTheta;
							ELSE
								alrTargetPos[LA_THETA] := alrTargetPos[LA_THETA] + sPartDataMMI.lrPartOffsetThetaLiftDrop;
								alrSecuredTarget[LA_X] := alrSecuredTarget[LA_X] + sPartDataMMI.lrPartOffsetXLiftDrop;
								alrSecuredTarget[LA_Y] := alrSecuredTarget[LA_Y] + sPartDataMMI.lrPartOffsetYLiftDrop;
							END_IF
							aeMoveRobotCommand[LA_THETA] := AC_MoveAtAbsPos;
							eReturnStep4SecureMove := SP_RunStp315;
							sCurrentState.eStep := SP_RunStp550;
						SP_RunStp315:
							IF eRobotXYTStatus = AS_InPosition THEN
								sCurrentState.eStep := SP_RunStp1;
							END_IF

						SP_RunStp330: (*Go to box position*)
							alrSecuredTarget[LA_X] := alrRobotPos[LTA_X,LTP_RejectBulkBox] + alrRobotOffset[LTA_X, iHead];
							alrSecuredTarget[LA_Y] :=alrRobotPos[LTA_Y,LTP_RejectBulkBox] + alrRobotOffset[LTA_Y, iHead];
							alrTargetPos[LA_THETA] := alrRobotPos[LTA_THETA,LTP_TableSideALayering1] + alrRobotOffset[LTA_THETA, iHead];
							aeMoveRobotCommand[LA_THETA] := AC_MoveAtAbsPos;
							eReturnStep4SecureMove := SP_RunStp331;
							sCurrentState.eStep := SP_RunStp550;
						SP_RunStp331:
							IF eRobotXYTStatus = AS_InPosition THEN
								sCurrentState.eStep := SP_RunStp1;
							END_IF

						SP_RunStp400 : (*move XYZ to safe *)
							IF (eLift1RunStatus = RS_WaitRequest OR sLift1RunData.eLiftPos = LP_OpenDrawer) AND (eLift2RunStatus = RS_WaitRequest OR sLift2RunData.eLiftPos = LP_OpenDrawer) THEN
								IF eLift1RunStatus = RS_WaitRequest THEN eLift1RunCmd := RCL_MoveToOpenDrawer; END_IF
								IF eLift2RunStatus = RS_WaitRequest THEN eLift2RunCmd := RCL_MoveToOpenDrawer; END_IF
								bMovePlateTakerDown := FALSE;
								sCurrentState.eStep := SP_RunStp401;
							END_IF
						SP_RunStp401 :
							IF (bPlateTakerIsUp) THEN
								(* Move Z to Safe *)
								alrTargetPos[LA_Z1] := alrSecuredSafeZPos[0] (*alrSafePos[LA_Z1]*);
								alrTargetPos[LA_Z2] := alrSecuredSafeZPos[1] (*alrSafePos[LA_Z2]*);
								aeMoveRobotCommand[LA_Z1] := AC_MoveAtAbsPos;
								aeMoveRobotCommand[LA_Z2] := AC_MoveAtAbsPos;
								sCurrentState.eStep := SP_RunStp402;
							END_IF
						SP_RunStp402:
							(* Wait until we are up *)
							IF ((aTRobotAxis[LA_Z1].eCurrentState = AS_InPosition) OR
									(bUse103171OptimB5MoveOnPreSafeZ AND  (aTRobotAxis[LA_Z1].lrCurrentPos < (alrSecuredSafeZPos[0]+lrPreSafeTolerance)))) AND
									((aTRobotAxis[LA_Z2].eCurrentState = AS_InPosition) OR
									(bUse103171OptimB5MoveOnPreSafeZ AND  (aTRobotAxis[LA_Z2].lrCurrentPos < (alrSecuredSafeZPos[1]+lrPreSafeTolerance)))) THEN
								(* Move X/ Y to Safe *)
								alrSecuredTarget[LA_X] := alrSafePos[LA_X];
								alrSecuredTarget[LA_Y] := alrSafePos[LA_Y];
								eReturnStep4SecureMove := SP_RunStp403;
								sCurrentState.eStep := SP_RunStp550;
							END_IF
						SP_RunStp403:
							IF aTRobotAxis[LA_X].eCurrentState =  AS_InPosition AND aTRobotAxis[LA_Y].eCurrentState =  AS_InPosition AND sLift1RunData.eLiftPos = LP_OpenDrawer AND sLift2RunData.eLiftPos = LP_OpenDrawer THEN
								sCurrentState.eStep := SP_RunStp1;
							END_IF
						SP_RunStp410 : (*Scan plate*)
							FOR i := 0 TO C_MAX_NB_OF_PARTS_ON_PLATE DO
								aTScanResult[i].bPresent := FALSE;
								aTScanResult[i].bValid := FALSE;
								aTScanResult[i].lrScore := -1;
								aTScanResult[i].lrTheta := 0;
								aTScanResult[i].lrX := 0;
								aTScanResult[i].lrY := 0;
							END_FOR
							sRunData.iCurrentScanOK := 0;
							sRunData.iCurrentScanTotal := 0;
							CASE sRunData.eModule OF
								LMP_Lift1:
									eScanPos := LTP_Lift1;
									sCurrentState.eStep := SP_RunStp411;
								LMP_Lift2:
									eScanPos := LTP_Lift2;
									sCurrentState.eStep := SP_RunStp412;
								LMP_Reject:
									eScanPos := LTP_Reject;
									sCurrentState.eStep := SP_RunStp413;
							END_CASE
						SP_RunStp411: (* Check Lift Status*)
							IF eLift1RunStatus = RS_WaitRequest THEN
								CASE sLift1RunData.eLiftPos OF
									LP_OnPlate:
										iPlatePos := 0;
										sCurrentState.eStep := SP_RunStp415;
									LP_Full,LP_Empty:
										bLift1NeedsPlate := TRUE;
										eLift1RunCmd := RCL_MoveToOpenDrawer;
									ELSE
										eLift1RunCmd := RCL_MoveToPlate;
								END_CASE
							END_IF
						SP_RunStp412: (* Check Lift Status*)
							IF eLift2RunStatus = RS_WaitRequest THEN
								CASE sLift2RunData.eLiftPos OF
									LP_OnPlate:
										iPlatePos := 0;
										sCurrentState.eStep := SP_RunStp415;
									LP_Full,LP_Empty:
										bLift2NeedsPlate := TRUE;
										eLift2RunCmd := RCL_MoveToOpenDrawer;
									ELSE
										eLift2RunCmd := RCL_MoveToPlate;
								END_CASE
							END_IF
						SP_RunStp413: (* Check Reject Status*)
							IF eRejectRunStatus = RS_WaitRequest THEN
								CASE sRejectRunData.eRejectStatus OF
									RS_Ready:
										eRejectRunCmd := RCR_LockDrawer;
									RS_Locked:
										iPlatePos := 0;
										sCurrentState.eStep := SP_RunStp415;
									ELSE
										bRejectNeedsPlate := TRUE;
										eRejectRunCmd := RCR_OpenDrawer;
								END_CASE
							END_IF
						SP_RunStp415: (*Scan Vision Part Position *)
							alrSecuredTarget[LA_X] := alrRobotPos[LTA_X,eScanPos] + alrRobotOffset[LTA_X, LTO_Vision] + alrLiftCalibrationOffset[eScanPos,LTA_X]  - sPlateData.alrPartOnPlate[iPlatePos].lrX ;
							alrSecuredTarget[LA_Y] :=  alrRobotPos[LTA_Y,eScanPos] + alrRobotOffset[LTA_Y, LTO_Vision] + alrLiftCalibrationOffset[eScanPos,LTA_Y] - sPlateData.alrPartOnPlate[iPlatePos].lrY ;
							TVisionWaitStab(IN := FALSE);
							eReturnStep4SecureMove := SP_RunStp416;
							sCurrentState.eStep := SP_RunStp550;
						SP_RunStp416:
							IF eRobotXYTStatus = AS_InPosition THEN
								TVisionWaitStab(IN := TRUE, PT := TVisionWaitStabTime);
								IF TVisionWaitStab.Q THEN
									eVisionRunCmd := RCV_GrabImage;
									sCurrentState.eStep := SP_RunStp417;
								END_IF
							END_IF
						SP_RunStp417:
							IF eVisionRunStatus = RS_WaitRequest THEN
								sRunDataVision.iUseModel := sRunData.iScanModel;
								eVisionRunCmd := RCV_AnalyseImage;
								sCurrentState.eStep := SP_RunStp419;
							END_IF
						SP_RunStp419: (* Check for part *)
							IF eVisionRunStatus = RS_WaitRequest THEN
								aTScanResult[iPlatePos] := sRunDataVision.TVisionPartData;
								iPlatePos := iPlatePos + 1;
								IF sRunDataVision.TVisionPartData.bValid THEN
									sRunData.iCurrentScanOK := sRunData.iCurrentScanOK + 1;
								END_IF
								sRunData.iCurrentScanTotal := sRunData.iCurrentScanTotal + 1;
								IF (iPlatePos < sPlateData.iNbPartOnPlate) THEN
									sCurrentState.eStep := SP_RunStp415;
								ELSE
									sCurrentState.eStep := SP_RunStp420;
								END_IF
							END_IF
						SP_RunStp420: (* Unlock Reject if needed *)
							IF sRunData.eModule = LMP_Reject AND eRejectRunStatus = RS_WaitRequest AND sRejectRunData.eRejectStatus=RS_Locked THEN
								eRejectRunCmd := RCR_UnlockDrawer;
							END_IF
							sCurrentState.eStep := SP_RunStp1;
						SP_RunStp500: (* Measure Z position on lift *)
							iZSensorPositionScan := 0;
							lrPartX := sPlateData.alrPartOnPlate[0].lrX;
							lrPartY := sPlateData.alrPartOnPlate[0].lrY;
							sCurrentState.eStep := SP_RunStp501;
						SP_RunStp501:
							alrSecuredTarget[LA_X] := alrRobotPos[LTA_X,eScanPos] + alrRobotOffset[LTA_X, LTO_ZSensor] + alrLiftCalibrationOffset[eScanPos,LTA_X]  -  lrPartX - sPartDataMMI.alrSensorZOffset[iZSensorPositionScan].lrX;
							alrSecuredTarget[LA_Y] :=alrRobotPos[LTA_Y,eScanPos] + alrRobotOffset[LTA_Y, LTO_ZSensor] + alrLiftCalibrationOffset[eScanPos,LTA_Y] - lrPartY - sPartDataMMI.alrSensorZOffset[iZSensorPositionScan].lrY;
							TSensorZWaitStab(IN := FALSE);
							sCurrentState.bWaitStep := TRUE;
							eReturnStep4SecureMove := SP_RunStp502;
							sCurrentState.eStep := SP_RunStp550;
						SP_RunStp502:
							IF eRobotXYTStatus = AS_InPosition THEN
								TSensorZWaitStab(IN := TRUE, PT := TSensorZWaitStabTime);
								IF TSensorZWaitStab.Q THEN
									IF TSensorMeasure.bInputOutOfRange THEN
										bZSensorOutOfRangeError := TRUE;
									END_IF
									lrZSensorPosition[iZSensorPositionScan] := TSensorMeasure.lrValue;
									IF iZSensorPositionScan = 0 AND (sPartDataMMI.alrSensorZOffset[1].lrX<>0 OR sPartDataMMI.alrSensorZOffset[1].lrY<>0) THEN
										iZSensorPositionScan := iZSensorPositionScan + 1;
										lrPartX := sPlateData.alrPartOnPlate[sPlateData.iNbPartOnPlate-1].lrX;
										lrPartY := sPlateData.alrPartOnPlate[sPlateData.iNbPartOnPlate-1].lrY;
										sCurrentState.eStep := SP_RunStp501;
									ELSE
										sCurrentState.eStep := SP_RunStp503;
									END_IF
								END_IF
							END_IF
						SP_RunStp503:
							IF iZSensorPositionScan = 1 THEN
								(* We used two position, mean the value *)
								alrZLiftPos[eScanPos] := (lrZSensorPosition[0] + lrZSensorPosition[1]) / 2;
							ELSE
								(* Only one position, use the first one then *)
								alrZLiftPos[eScanPos] := lrZSensorPosition[0];
							END_IF
							sCurrentState.eStep := eReturnStepMeasureZLift;
						SP_RunStp550:	// Move XY without entering unsecured area
							// Check if we enter area on Y
							IF (alrSecuredTarget[LA_Y] > alrUnsecuredArea[0,LA_Y]) AND (aTRobotAxis[LA_Y].lrCurrentPos < (alrUnsecuredArea[0,LA_Y] - lrSafeTolerance)) THEN
								// We have to go around area coming from neg
								iSecuredIndexFirst := 0;
								iSecuredIndexSecond := 1;
								sCurrentState.eStep := SP_RunStp555;
							ELSIF (alrSecuredTarget[LA_Y] < alrUnsecuredArea[1,LA_Y]) AND (aTRobotAxis[LA_Y].lrCurrentPos > (alrUnsecuredArea[1,LA_Y] + lrSafeTolerance )) THEN
								// We have to go around area coming from pos
								iSecuredIndexFirst := 1;
								iSecuredIndexSecond := 0;
								sCurrentState.eStep := SP_RunStp555;
							ELSE
								alrTargetPos[LA_X] := alrSecuredTarget[LA_X];
								alrTargetPos[LA_Y] := alrSecuredTarget[LA_Y];
								aeMoveRobotCommand[LA_X] := AC_MoveAtAbsPos;
								aeMoveRobotCommand[LA_Y] := AC_MoveAtAbsPos;
								sCurrentState.eStep := SP_RunStp599;
							END_IF
						SP_RunStp555:	// Go around area
							IF alrTargetPos[LA_Z1] <> alrSecuredSafeZPos[0] THEN
								alrTargetPos[LA_Z1] := alrSecuredSafeZPos[0];
								aeMoveRobotCommand[LA_Z1] := AC_MoveAtAbsPos;
							END_IF
							IF alrTargetPos[LA_Z2] <> alrSecuredSafeZPos[1] THEN
								alrTargetPos[LA_Z2] := alrSecuredSafeZPos[1];
								aeMoveRobotCommand[LA_Z2] := AC_MoveAtAbsPos;
							END_IF
							IF (alrSecuredTarget[LA_X] < alrUnsecuredArea[1,LA_X]) THEN // HFO
							//IF ((alrSecuredTarget[LA_X] - alrUnsecuredArea[1,LA_X]) * ((alrUnsecuredArea[1,LA_X] + lrSafeTolerance) - aTRobotAxis[LA_X].lrCurrentPos)) < 0 THEN
								alrTargetPos[LA_X] := alrUnsecuredArea[1,LA_X] + lrSafeTolerance;
								toto := FALSE;
							ELSE
								alrTargetPos[LA_X] := alrSecuredTarget[LA_X];
								toto := TRUE;
							END_IF
							alrTargetPos[LA_Y] := alrUnsecuredArea[iSecuredIndexFirst,LA_Y] + iSecuredIndexFirst * lrSafeTolerance - iSecuredIndexSecond * lrSafeTolerance;
							aeMoveRobotCommand[LA_X] := AC_MoveAtAbsPos;
							aeMoveRobotCommand[LA_Y] := AC_MoveAtAbsPos;
							sCurrentState.eStep := SP_RunStp556;
						SP_RunStp556:	
//							IF eRobotXYTStatus = AS_InPosition THEN
							IF (aTRobotAxis[LA_Z1].eCurrentState = AS_InPosition)
								AND (aTRobotAxis[LA_Z2].eCurrentState = AS_InPosition)
								AND ABS(alrTargetPos[LA_X] - aTRobotAxis[LA_X].lrCurrentPos) < 1 THEN
								alrTargetPos[LA_Y] := alrUnsecuredArea[iSecuredIndexSecond,LA_Y] + iSecuredIndexSecond * lrSafeTolerance - iSecuredIndexFirst * lrSafeTolerance;
								aeMoveRobotCommand[LA_Y] := AC_MoveAtAbsPos;
								sCurrentState.eStep := SP_RunStp557;
							END_IF
						SP_RunStp557:	
//							IF eRobotXYTStatus = AS_InPosition THEN
							IF 	ABS(alrTargetPos[LA_Y] - aTRobotAxis[LA_Y].lrCurrentPos) < 5
								AND ABS(alrTargetPos[LA_X] - aTRobotAxis[LA_X].lrCurrentPos) < 5 THEN
								alrTargetPos[LA_X] := alrSecuredTarget[LA_X];
								alrTargetPos[LA_Y] := alrSecuredTarget[LA_Y];
								aeMoveRobotCommand[LA_X] := AC_MoveAtAbsPos;
								aeMoveRobotCommand[LA_Y] := AC_MoveAtAbsPos;
								sCurrentState.eStep := SP_RunStp599;
							END_IF
						SP_RunStp599:	
							IF eRobotXYTStatus = AS_InPosition THEN
								// return back to process
								sCurrentState.eStep := eReturnStep4SecureMove;
							END_IF
					END_CASE
				END_IF
			MS_Manual :	// Manual Mode to move axis indepedentely
				TManualCmd.eTableSide := eTableSide;	// Position of the table : A, B or Moving
				// Control of safe position of Z_1 and Z_2
				TManualCmd.bAxisZSafe[0] := (aTRobotAxis[LA_Z1].lrCurrentPos < (alrSafePos[LA_Z1]+lrSafeTolerance)) AND ((aTRobotAxis[LA_Z1].eCurrentState = AS_InPosition) OR (aTRobotAxis[LA_Z1].eCurrentState = AS_PowerOff)) AND (aTRobotAxis[LA_Z1].bAxisHomed);
				TManualCmd.bAxisZSafe[1] := (aTRobotAxis[LA_Z2].lrCurrentPos < (alrSafePos[LA_Z2]+lrSafeTolerance)) AND ((aTRobotAxis[LA_Z2].eCurrentState = AS_InPosition) OR (aTRobotAxis[LA_Z1].eCurrentState = AS_PowerOff)) AND (aTRobotAxis[LA_Z1].bAxisHomed);;
				
				iRobotPosition := UINT_TO_INT(TManualCmd.wRobotPos AND 15);
				iRobotOffset := UINT_TO_INT(SHR(TManualCmd.wRobotPos AND 2#1111_1111_1111_0000(*NOT 15*),4));

				bManualZIsSafe :=  (aTRobotAxis[LA_Z1].lrCurrentPos < (alrSafePos[LA_Z1]+lrSafeTolerance)) AND (aTRobotAxis[LA_Z2].lrCurrentPos < (alrSafePos[LA_Z2]+lrSafeTolerance))
								(*AND ((aTRobotAxis[LA_Z1].eCurrentState = AS_InPosition) OR (aTRobotAxis[LA_Z1].eCurrentState = AS_PowerOff))
								AND ((aTRobotAxis[LA_Z2].eCurrentState = AS_InPosition)  OR (aTRobotAxis[LA_Z2].eCurrentState = AS_PowerOff))*)
								AND (aTRobotAxis[LA_Z1].bAxisHomed) AND (aTRobotAxis[LA_Z2].bAxisHomed) AND bPlateTakerIsUp;

				TManualCmd.TMovePlateTakerDown.Enable := ((aTRobotAxis[LA_X].eCurrentState = AS_InPosition) AND (aTRobotAxis[LA_Y].eCurrentState = AS_InPosition) AND bManualZIsSafe) OR NOT bPlateTakerIsUp ;
				TManualCmd.TSafe.Enable := TRUE;
				TManualCmd.TVisionCalibration.Enable := TRUE;
				FOR iAxis := 0 TO 4 DO
					iTeachedAxis := GetLoaderTeachedAxisFromAxis(iAxis);
					TManualCmd.TVisionCalibration.Enable := NOT bManInterlock AND TManualCmd.TVisionCalibration.Enable AND aTRobotAxis[iAxis].eCurrentState = AS_InPosition;
					TManualCmd.TSafe.Enable := TManualCmd.TSafe.Enable AND ((aTRobotAxis[iAxis].eCurrentState = AS_InPosition) OR  (aTRobotAxis[iAxis].eCurrentState = AS_PowerOff) OR  (aTRobotAxis[iAxis].eCurrentState = AS_OnLimitNeg)  OR  (aTRobotAxis[iAxis].eCurrentState = AS_NotHomed));
					TManualCmd.aTAxis[iAxis].Home.Enable := NOT (bManInterlock AND (NOT INT_TO_UINT(iAxis) = 2 OR NOT INT_TO_UINT(iAxis) = 3 OR NOT INT_TO_UINT(iAxis) = 4)) AND ((aTRobotAxis[iAxis].eCurrentState = AS_InPosition) OR (aTRobotAxis[iAxis].eCurrentState = AS_NotHomed) OR (aTRobotAxis[iAxis].eCurrentState = AS_OnLimitNeg)) AND iManMoveAxis=iManMoveAxisNone
															AND NOT((INT_TO_UINT(iAxis) > 1) AND (aTRobotAxis[LA_X].lrCurrentPos > alrUnsecuredArea[0,LA_X]+ lrSafeTolerance) AND (aTRobotAxis[LA_X].lrCurrentPos < alrUnsecuredArea[1,LA_X] - lrSafeTolerance) AND (aTRobotAxis[LA_Y].lrCurrentPos > alrUnsecuredArea[0,LA_Y]+ lrSafeTolerance) AND (aTRobotAxis[LA_Y].lrCurrentPos < alrUnsecuredArea[1,LA_Y] - lrSafeTolerance));
					//TManualCmd.aTAxis[iAxis].Home.Enable := NOT (bManInterlock AND iAxis > 1) AND ((aTRobotAxis[iAxis].eCurrentState = AS_InPosition) OR (aTRobotAxis[iAxis].eCurrentState = AS_NotHomed) OR (aTRobotAxis[iAxis].eCurrentState = AS_OnLimitNeg)) AND iManMoveAxis=iManMoveAxisNone;

					(*TManualCmd.aTAxis[iAxis].Home.Enable := ((aTRobotAxis[iAxis].eCurrentState = AS_InPosition) OR (aTRobotAxis[iAxis].eCurrentState = AS_NotHomed) OR (aTRobotAxis[iAxis].eCurrentState = AS_OnLimitNeg)) AND iManMoveAxis=iManMoveAxisNone;
					IF iAxis < 3 THEN
						TManualCmd.aTAxis[iAxis].Home.Enable := TManualCmd.aTAxis[iAxis].Home.Enable AND NOT bManInterlock;
					END_IF*)

					TManualCmd.aTAxis[iAxis].MoveBw.Enable := NOT bManInterlock AND iManMoveAxis=iManMoveAxisNone AND (aTRobotAxis[iAxis].eCurrentState = AS_InPosition) AND ((aTRobotAxis[iAxis].lrCurrentPos - alrJogStep[iAxis] >= aTRobotAxis[iAxis].lrMinPos) OR NOT aTRobotAxis[iAxis].bMinPosMonitoring);
					TManualCmd.aTAxis[iAxis].MoveFw.Enable := NOT bManInterlock AND iManMoveAxis=iManMoveAxisNone AND (aTRobotAxis[iAxis].eCurrentState = AS_InPosition) AND ((aTRobotAxis[iAxis].lrCurrentPos + alrJogStep[iAxis] <= aTRobotAxis[iAxis].lrMaxPos) OR NOT aTRobotAxis[iAxis].bMaxPosMonitoring);


					TManualCmd.aTAxisPos[iAxis].TeachedPos := alrRobotPos[iTeachedAxis, iRobotPosition] + alrRobotOffset[iTeachedAxis,iRobotOffset];
					IF (iRobotOffset = LTO_Plate) AND (iRobotPosition = LTP_Lift1) THEN
						TManualCmd.aTAxisPos[LA_X].TeachedPos := alrRobotPos[LTA_X,LTP_Lift1] +alrRobotOffset[LTA_X, LTO_Plate] + alrLiftCalibrationOffset[LTP_Lift1,LTA_X] - sPlateData.alrTakePlatePos.lrX;
						TManualCmd.aTAxisPos[LA_Y].TeachedPos := alrRobotPos[LTA_Y,LTP_Lift1] +alrRobotOffset[LTA_Y, LTO_Plate] + alrLiftCalibrationOffset[LTP_Lift1,LTA_Y] - sPlateData.alrTakePlatePos.lrY;
					END_IF
					TManualCmd.aTAxisPos[iAxis].MoveToTeach.Enable := NOT bManInterlock AND iManMoveAxis=iManMoveAxisNone AND (aTRobotAxis[iAxis].eCurrentState = AS_InPosition) AND
							(( TManualCmd.aTAxisPos[iAxis].TeachedPos >= aTRobotAxis[iAxis].lrMinPos) OR NOT aTRobotAxis[iAxis].bMinPosMonitoring) AND
							((TManualCmd.aTAxisPos[iAxis].TeachedPos <= aTRobotAxis[iAxis].lrMaxPos) OR NOT aTRobotAxis[iAxis].bMaxPosMonitoring);
					TManualCmd.aTAxis[iAxis].CurrentPos := aTRobotAxis[iAxis].lrCurrentPos;
					alrRobotSpeed[iAxis] := aTRobotAxis[iAxis].lrManualSpeed;
				END_FOR
				TManualCmd.TMoveVision2Table.Enable := bManualZIsSafe;
				TManualCmd.TMoveVision2Lift.Enable := bManualZIsSafe;
				IF NOT bManualZIsSafe THEN
					TManualCmd.aTAxis[LA_X].Home.Enable := FALSE;
					TManualCmd.aTAxis[LA_Y].Home.Enable := FALSE;
					IF alrJogStep[LA_X] > lrMaxXYMoveAllowed-0.1 THEN
						TManualCmd.aTAxis[LA_X].MoveBw.Enable := FALSE;
						TManualCmd.aTAxis[LA_X].MoveFw.Enable := FALSE;
					END_IF
					IF alrJogStep[LA_Y] > lrMaxXYMoveAllowed-0.1 THEN
						TManualCmd.aTAxis[LA_Y].MoveBw.Enable := FALSE;
						TManualCmd.aTAxis[LA_Y].MoveFw.Enable := FALSE;
					END_IF
					IF alrJogStep[LA_Z1] > lrMaxXYMoveAllowed-0.1 THEN
						TManualCmd.aTAxis[LA_Z1].MoveFw.Enable := FALSE;
					END_IF
					IF alrJogStep[LA_Z2] > lrMaxXYMoveAllowed-0.1 THEN
						TManualCmd.aTAxis[LA_Z2].MoveFw.Enable := FALSE;
					END_IF
					TManualCmd.aTAxisPos[LA_X].MoveToTeach.Enable := TManualCmd.aTAxisPos[LA_X].MoveToTeach.Enable AND ABS(TManualCmd.aTAxisPos[LA_X].TeachedPos-aTRobotAxis[LA_X].lrCurrentPos) < lrMaxXYMoveAllowed-0.1;
					TManualCmd.aTAxisPos[LA_Y].MoveToTeach.Enable := TManualCmd.aTAxisPos[LA_Y].MoveToTeach.Enable AND ABS(TManualCmd.aTAxisPos[LA_Y].TeachedPos-aTRobotAxis[LA_Y].lrCurrentPos) < lrMaxXYMoveAllowed-0.1;
				END_IF
				FOR i:= 0 TO 1 DO
					TManualCmd.alrVaccumValue[i] := aTHeadVacuum[i].lrVacuum;
				END_FOR
				
				TManualCmd.lrSensorMeasure := TSensorMeasure.lrValue;
				TManualCmd.TZSensorTeach.Enable := (eTableSide = TS_A) AND NOT TSensorMeasure.bInputOutOfRange;

				bManInterlockLiftOut := NOT bManualZIsSafe;
				bManInterlockOut := NOT ((aTRobotAxis[LA_Z1].lrCurrentPos < (alrSafePos[LA_Z1]+lrSafeTolerance)) AND (aTRobotAxis[LA_Z2].lrCurrentPos < (alrSafePos[LA_Z2]+lrSafeTolerance)) AND
								 (*(aTRobotAxis[LA_X].lrCurrentPos < (alrSafePos[LA_X]+lrSafeTolerance)) AND (aTRobotAxis[LA_Y].lrCurrentPos < (alrSafePos[LA_Y]+lrSafeTolerance)) AND*)
								(*AND ((aTRobotAxis[LA_Z1].eCurrentState = AS_InPosition) OR (aTRobotAxis[LA_Z1].eCurrentState = AS_PowerOff))
								AND ((aTRobotAxis[LA_Z2].eCurrentState = AS_InPosition)  OR (aTRobotAxis[LA_Z2].eCurrentState = AS_PowerOff))*)
								(*(aTRobotAxis[LA_X].bAxisHomed) AND (aTRobotAxis[LA_Y].bAxisHomed) AND*)
								(aTRobotAxis[LA_Z1].bAxisHomed) AND (aTRobotAxis[LA_Z2].bAxisHomed) AND bPlateTakerIsUp);
				CASE sCurrentState.eStep OF
					SP_ManualStp0 :
						TManualCmd.TPlateVacuum.Enable := TRUE;
						TManualCmd.THead1Vacuum.Enable := TRUE;
						TManualCmd.THead2Vacuum.Enable := TRUE;
						TManualCmd.TPlateVacuum.Activate := bEnablePlateVacuum;
						TManualCmd.TMovePlateTakerDown.Activate := bMovePlateTakerDown;
						TManualCmd.THead1Vacuum.Activate := abEnableHeadVacuum[0];
						TManualCmd.THead2Vacuum.Activate := abEnableHeadVacuum[1];
						FOR iAxis := 0 TO 4 DO
							TManualCmd.aTAxis[iAxis].Home.Activate := FALSE;
							TManualCmd.aTAxis[iAxis].MoveFw.Activate := FALSE;
							TManualCmd.aTAxis[iAxis].MoveBw.Activate := FALSE;
							TManualCmd.aTAxisPos[iAxis].MoveToTeach.Activate := FALSE;
							TManualCmd.aTAxisPos[iAxis].Teach := FALSE;
							TManualCmd.aTAxisPos[iAxis].MoveToTeach.Enable := FALSE;
							TManualCmd.aTAxis[iAxis].JogStep := alrJogStep[iAxis];
						END_FOR
						FOR i:= 0 TO 1 DO
							TManualCmd.alrVaccumThershold[i] := alrVacuumThreshold[i];
						END_FOR
						TManualCmd.TVisionCalibration.Activate := FALSE;
						TManualCmd.TSafe.Activate := FALSE;
						TManualCmd.TZSensorTeach.Activate := FALSE;
						 iManMoveAxis:=iManMoveAxisNone;
						TManualCmd.TAspirationBrush.Enable := TRUE;
						TManualCmd.TAspirationBrush.Activate := bAspirationBrushOn;
						TManualCmd.lrSensorAdjust := lrSensorAdjust;
						TManualCmd.TMoveVision2Table.Activate := FALSE;
						TManualCmd.TMoveVision2Lift.Activate := FALSE;
						sCurrentState.eStep := SP_ManualStp1;
					SP_ManualStp1 :
						IF bStopReq THEN
							sCurrentState.eStatus := MS_Stopped;
						ELSE
							FOR iAxis := 0 TO 4 DO
								iTeachedAxis := GetLoaderTeachedAxisFromAxis(iAxis);
								IF TManualCmd.aTAxisPos[iAxis].Teach THEN
									TManualCmd.aTAxisPos[iAxis].Teach := FALSE; (* change here the learning teach *)
									IF (iRobotOffset = LTO_Z1) THEN
										alrRobotOffset[iTeachedAxis,iRobotOffset] := 0;
										alrRobotPos[iTeachedAxis, iRobotPosition] := aTRobotAxis[iAxis].lrCurrentPos;
										iTeachedModeDebug := 0;
									ELSIF (iRobotOffset <> LTO_Plate) THEN (* Plate position are hardcoded, cannot be teached *)
										alrRobotOffset[iTeachedAxis, iRobotOffset] := aTRobotAxis[iAxis].lrCurrentPos - alrRobotPos[iTeachedAxis, iRobotPosition];
										iTeachedModeDebug := 1;
									END_IF
								END_IF
								IF (alrJogStep[iAxis] <> TManualCmd.aTAxis[iAxis].JogStep) THEN
									alrJogStep[iAxis] := TManualCmd.aTAxis[iAxis].JogStep;
								END_IF
								IF TManualCmd.aTAxisPos[iAxis].MoveToTeach.Activate AND iManMoveAxis=iManMoveAxisNone THEN
									alrTargetPos[iAxis] := TManualCmd.aTAxisPos[iAxis].TeachedPos;
									iManMoveAxis := iAxis;
									sCurrentState.eStep := SP_ManualStp10;
								END_IF
								IF TManualCmd.aTAxis[iAxis].MoveFw.Activate AND iManMoveAxis=iManMoveAxisNone THEN
									alrTargetPos[iAxis] := aTRobotAxis[iAxis].lrCurrentPos + alrJogStep[iAxis];
									iManMoveAxis := iAxis;
									sCurrentState.eStep := SP_ManualStp10;
								END_IF
								IF TManualCmd.aTAxis[iAxis].MoveBw.Activate AND iManMoveAxis=iManMoveAxisNone THEN
									alrTargetPos[iAxis] := aTRobotAxis[iAxis].lrCurrentPos - alrJogStep[iAxis];
									iManMoveAxis := iAxis;
									sCurrentState.eStep := SP_ManualStp10;
								END_IF
								IF TManualCmd.aTAxis[iAxis].Home.Activate AND  iManMoveAxis=iManMoveAxisNone THEN
									iManMoveAxis := iAxis;
									sCurrentState.eStep := SP_ManualStp20;
								END_IF
							END_FOR
							FOR i:= 0 TO 1 DO
								IF TManualCmd.alrVaccumThershold[i] <> alrVacuumThreshold[i] THEN
									alrVacuumThreshold[i] := TManualCmd.alrVaccumThershold[i];
								END_IF
							END_FOR
							IF TManualCmd.TSafe.Activate AND  iManMoveAxis=iManMoveAxisNone THEN
								TManualCmd.TSafe.Activate := FALSE;
								iManMoveAxis:=LA_X;
								sCurrentState.eStep := SP_ManualStp30;
							END_IF
							IF TManualCmd.TVisionCalibration.Activate AND  iManMoveAxis=iManMoveAxisNone THEN
								TManualCmd.TVisionCalibration.Activate := FALSE;
								iManMoveAxis:=LA_X;
								sCurrentState.eStep := SP_ManualStp50;
							END_IF
							IF (lrSensorAdjust <> TManualCmd.lrSensorAdjust) THEN
								lrSensorAdjust :=  TManualCmd.lrSensorAdjust;
							END_IF
							IF TManualCmd.TZSensorTeach.Activate THEN
								TManualCmd.TZSensorTeach.Activate := FALSE;
								lrSensorAdjust := 0 - (TSensorMeasure.lrValue - lrSensorAdjust);
								TManualCmd.lrSensorAdjust := lrSensorAdjust;
							END_IF
							IF TManualCmd.TMoveVision2Table.Activate  AND  iManMoveAxis=iManMoveAxisNone THEN
								TManualCmd.TMoveVision2Table.Activate := FALSE;
								iManMoveAxis:=LA_X;
								alrTargetPos[LA_X] := alrRobotPos[LTA_X,LTP_TableSideALayering1]  -  sPartDataMMI.alrPartOffsetLayering[sRunData.iLayringOffsetPos].lrX + alrRobotOffset[LTA_X, LTO_Vision];
								alrTargetPos[LA_Y] :=  alrRobotPos[LTA_Y,LTP_TableSideALayering1]  + sPartDataMMI.alrPartOffsetLayering[sRunData.iLayringOffsetPos].lrY + alrRobotOffset[LTA_Y, LTO_Vision];
								sCurrentState.eStep := SP_ManualStp70;
							END_IF
							IF TManualCmd.TMoveVision2Lift.Activate  AND  iManMoveAxis=iManMoveAxisNone THEN
								TManualCmd.TMoveVision2Lift.Activate := FALSE;
								iManMoveAxis:=LA_X;
								alrTargetPos[LA_X] := alrRobotPos[LTA_X,LTP_Lift1] + alrRobotOffset[LTA_X, LTO_Vision] + alrLiftCalibrationOffset[LTP_Lift1,LTA_X]  - sPlateData.alrPartOnPlate[TManualCmd.wMoveVision2LiftPos-1].lrX ;
								alrTargetPos[LA_Y] :=  alrRobotPos[LTA_Y,LTP_Lift1] + alrRobotOffset[LTA_Y, LTO_Vision] + alrLiftCalibrationOffset[LTP_Lift1,LTA_Y] - sPlateData.alrPartOnPlate[TManualCmd.wMoveVision2LiftPos-1].lrY ;
								sCurrentState.eStep := SP_ManualStp70;
							END_IF
						END_IF
					SP_ManualStp10: (* Do the movement *)
						aeMoveRobotCommand[iManMoveAxis] := AC_MoveAtAbsPos;
						sCurrentState.eStep := SP_ManualStp11;
					SP_ManualStp11: (* Wait until position is reached *)
						CASE aTRobotAxis[iManMoveAxis].eCurrentState OF
							AS_InPosition, AS_InError:
								FOR iAxis := 0 TO 4 DO
									TManualCmd.aTAxis[iAxis].Home.Activate := FALSE;
									TManualCmd.aTAxis[iAxis].MoveFw.Activate := FALSE;
									TManualCmd.aTAxis[iAxis].MoveBw.Activate := FALSE;
									TManualCmd.aTAxisPos[iAxis].MoveToTeach.Activate := FALSE;
								END_FOR
								 iManMoveAxis:=iManMoveAxisNone;
								sCurrentState.eStep := SP_ManualStp1;
						END_CASE
					SP_ManualStp20 : (* Init axis *)
						aeMoveRobotCommand[iManMoveAxis] := AC_Home;
						sCurrentState.eStep := SP_ManualStp21;
					SP_ManualStp21 : (* Rotate the turn over to go to index position *)
						CASE aTRobotAxis[iManMoveAxis].eCurrentState OF
							AS_InPosition, AS_InError:
								FOR iAxis := 0 TO 4 DO
									TManualCmd.aTAxis[iAxis].Home.Activate := FALSE;
									TManualCmd.aTAxis[iAxis].MoveFw.Activate := FALSE;
									TManualCmd.aTAxis[iAxis].MoveBw.Activate := FALSE;
								END_FOR
								 iManMoveAxis:=iManMoveAxisNone;
								sCurrentState.eStep := SP_ManualStp1;
						END_CASE
					SP_ManualStp30: (* Move taker up *)
						TManualCmd.TMovePlateTakerDown.Activate := FALSE;
						IF bPlateTakerIsUp THEN
							sCurrentState.eStep := SP_ManualStp31;
						ELSIF bJackError THEN
							iManMoveAxis:=iManMoveAxisNone;
							sCurrentState.eStep := SP_ManualStp1;
						END_IF
					SP_ManualStp31: (*Move  Z1 and Z2 to Limit*)
						aeMoveRobotCommand[LA_Z1] := AC_MoveLimitNeg;
						aeMoveRobotCommand[LA_Z2] := AC_MoveLimitNeg;
						sCurrentState.eStep := SP_ManualStp32;
					SP_ManualStp32:
						IF aTRobotAxis[LA_Z1].eCurrentState= AS_OnLimitNeg AND aTRobotAxis[LA_Z2].eCurrentState= AS_OnLimitNeg THEN
							sCurrentState.eStep := SP_ManualStp33;
						ELSIF (aTRobotAxis[LA_Z1].eCurrentState= AS_OnLimitNeg AND aTRobotAxis[LA_Z2].eCurrentState = AS_InError) OR
							    (aTRobotAxis[LA_Z1].eCurrentState= AS_InError AND aTRobotAxis[LA_Z2].eCurrentState = AS_OnLimitNeg) OR
							    (aTRobotAxis[LA_Z1].eCurrentState= AS_InError AND aTRobotAxis[LA_Z2].eCurrentState = AS_InError) THEN
							iManMoveAxis:=iManMoveAxisNone;
							sCurrentState.eStep := SP_ManualStp1;
						END_IF
					SP_ManualStp33: (* Init X/Y  *)
						aeMoveRobotCommand[LA_X] := AC_Init;
						aeMoveRobotCommand[LA_Y] := AC_Init;
						sCurrentState.eStep := SP_ManualStp34;
					SP_ManualStp34:
						IF aTRobotAxis[LA_X].eCurrentState= AS_InPosition AND aTRobotAxis[LA_Y].eCurrentState = AS_InPosition THEN
							sCurrentState.eStep := SP_ManualStp35;
						ELSIF (aTRobotAxis[LA_X].eCurrentState= AS_InPosition AND aTRobotAxis[LA_Y].eCurrentState = AS_InError) OR
							    (aTRobotAxis[LA_X].eCurrentState= AS_InError AND aTRobotAxis[LA_Y].eCurrentState = AS_InPosition) OR
							    (aTRobotAxis[LA_X].eCurrentState= AS_InError AND aTRobotAxis[LA_Y].eCurrentState = AS_InError) THEN
							iManMoveAxis:=iManMoveAxisNone;
							sCurrentState.eStep := SP_ManualStp1;
						END_IF
					SP_ManualStp35: (* Move X/Y *)
						aeMoveRobotCommand[LA_X] := AC_MoveAtAbsPos;
						aeMoveRobotCommand[LA_Y] := AC_MoveAtAbsPos;
						alrTargetPos[LA_X] := alrSafePos[LA_X];
						alrTargetPos[LA_Y] := alrSafePos[LA_Y];
						sCurrentState.eStep := SP_ManualStp36;
					SP_ManualStp36:
						IF aTRobotAxis[LA_X].eCurrentState= AS_InPosition AND aTRobotAxis[LA_Y].eCurrentState = AS_InPosition THEN
							sCurrentState.eStep := SP_ManualStp37;
						ELSIF (aTRobotAxis[LA_X].eCurrentState= AS_InPosition AND aTRobotAxis[LA_Y].eCurrentState = AS_InError) OR
							    (aTRobotAxis[LA_X].eCurrentState= AS_InError AND aTRobotAxis[LA_Y].eCurrentState = AS_InPosition) OR
							    (aTRobotAxis[LA_X].eCurrentState= AS_InError AND aTRobotAxis[LA_Y].eCurrentState = AS_InError) THEN
							iManMoveAxis:=iManMoveAxisNone;
							sCurrentState.eStep := SP_ManualStp1;
						END_IF
					SP_ManualStp37: (* Init Z1 and Z2*)
						aeMoveRobotCommand[LA_Z1] := AC_Init;
						aeMoveRobotCommand[LA_Z2] := AC_Init;
						sCurrentState.eStep := SP_ManualStp38;
					SP_ManualStp38:
						IF aTRobotAxis[LA_Z1].eCurrentState= AS_InPosition AND aTRobotAxis[LA_Z2].eCurrentState = AS_InPosition THEN
							sCurrentState.eStep := SP_ManualStp39;
						ELSIF (aTRobotAxis[LA_Z1].eCurrentState= AS_InPosition AND aTRobotAxis[LA_Z2].eCurrentState = AS_InError) OR
							    (aTRobotAxis[LA_Z1].eCurrentState= AS_InError AND aTRobotAxis[LA_Z2].eCurrentState = AS_InPosition) OR
							    (aTRobotAxis[LA_Z1].eCurrentState= AS_InError AND aTRobotAxis[LA_Z2].eCurrentState = AS_InError) THEN
							iManMoveAxis:=iManMoveAxisNone;
							sCurrentState.eStep := SP_ManualStp1;
						END_IF
					SP_ManualStp39: (* Move up Z1 and Z2 *)
						aeMoveRobotCommand[LA_Z1] := AC_MoveAtAbsPos;
						aeMoveRobotCommand[LA_Z2] := AC_MoveAtAbsPos;
						alrTargetPos[LA_Z1] := alrSafePos[LA_Z1];
						alrTargetPos[LA_Z2] := alrSafePos[LA_Z2];
						sCurrentState.eStep := SP_ManualStp40;
					SP_ManualStp40:
						IF (aTRobotAxis[LA_Z1].eCurrentState= AS_InPosition OR aTRobotAxis[LA_Z1].eCurrentState = AS_InError) AND
							    (aTRobotAxis[LA_Z2].eCurrentState= AS_InPosition OR aTRobotAxis[LA_Z2].eCurrentState = AS_InError) THEN
							iManMoveAxis:=iManMoveAxisNone;
							sCurrentState.eStep := SP_ManualStp1;
						END_IF
					SP_ManualStp50: (*Switch part for learning vision *)
						iHead := 0;
						alrTargetPos[LA_X] := alrRobotPos[LTA_X,LTP_TableSideALayering1] + alrRobotOffset[LTA_X, iHead];
						alrTargetPos[LA_Y] :=  alrRobotPos[LTA_Y,LTP_TableSideALayering1] + alrRobotOffset[LTA_Y, iHead];
						alrTargetPos[LA_THETA] := alrRobotPos[LTA_THETA,LTP_TableSideALayering1] + alrRobotOffset[LTA_THETA, iHead];
						ZPositionTakeGive := alrRobotPos[LTA_Z,LTP_TableSideALayering1] + alrRobotOffset[LTA_Z, iHead];
						alrTargetPos[LA_X] := alrTargetPos[LA_X]   -  sPartDataMMI.alrPartOffsetLayering[0].lrX;
						alrTargetPos[LA_Y] := alrTargetPos[LA_Y]  + sPartDataMMI.alrPartOffsetLayering[0].lrY;
						ZPositionTakeGive := ZPositionTakeGive + (lrCalibrationLayeringAndPartAndHeadHeight - sPartDataMMI.lrLayeringAndPartAndHeadHeight);
						aeMoveRobotCommand[LA_X] := AC_MoveAtAbsPos;
						aeMoveRobotCommand[LA_Y] := AC_MoveAtAbsPos;
						aeMoveRobotCommand[LA_THETA] := AC_MoveAtAbsPos;
						sCurrentState.eStep := SP_ManualStp51;
					SP_ManualStp51:
						IF eRobotXYTStatus = AS_InPosition THEN
							sCurrentState.eStep := SP_ManualStp52;
						END_IF
					SP_ManualStp52 :  (*Take Part*)
						ZPosition := ZPositionTakeGive + sPartDataMMI.lrPartOffsetZLayeringTake;
						alrTargetPos[LA_Z1+iHead] := ZPosition;
						aeMoveRobotCommand[LA_Z1+iHead] := AC_MoveAtAbsPos;
						sCurrentState.eStep := SP_ManualStp53;
					SP_ManualStp53 :  (*Movement done*)
						IF aTRobotAxis[LA_Z1+iHead].lrRemainingTimeToGo < 1 AND aTRobotAxis[LA_Z1+iHead].lrRemainingTimeToGo <> 0 THEN
							 TManualCmd.THead1Vacuum.Activate := TRUE;
						END_IF
						IF aTRobotAxis[LA_Z1+iHead].eCurrentState = AS_InPosition THEN
							 TManualCmd.THead1Vacuum.Activate := TRUE;
							sCurrentState.eStep := SP_ManualStp54;
						END_IF
					SP_ManualStp54 :
						(* Check if the part is on head *)
						IF aTHeadVacuum[iHead].bVacuumCorrect THEN
							alrTargetPos[LA_Z1+iHead] := alrSafePos[LA_Z1+iHead];
							aeMoveRobotCommand[LA_Z1+iHead] := AC_MoveAtAbsPos;
							sCurrentState.eStep := SP_ManualStp55;
						END_IF
					SP_ManualStp55 :  (*Movement done*)
						IF aTRobotAxis[LA_Z1+iHead].eCurrentState = AS_InPosition THEN
							iPlatePos := 0;
							iZSensorPositionScan := 0;
							sCurrentState.eStep := SP_ManualStp56;
						END_IF
					SP_ManualStp56:
						alrTargetPos[LA_X] := alrRobotPos[LTA_X,LTP_Lift2] + alrRobotOffset[LTA_X, LTO_ZSensor] + alrLiftCalibrationOffset[LTP_Lift2,LTA_X]  -  sPlateData.alrPartOnPlate[iPlatePos].lrX - sPartDataMMI.alrSensorZOffset[iZSensorPositionScan].lrX;
						alrTargetPos[LA_Y] :=alrRobotPos[LTA_Y,LTP_Lift2] + alrRobotOffset[LTA_Y, LTO_ZSensor] + alrLiftCalibrationOffset[LTP_Lift2,LTA_Y] - sPlateData.alrPartOnPlate[iPlatePos].lrY - sPartDataMMI.alrSensorZOffset[iZSensorPositionScan].lrY;
						aeMoveRobotCommand[LA_X] := AC_MoveAtAbsPos;
						aeMoveRobotCommand[LA_Y] := AC_MoveAtAbsPos;
						TSensorZWaitStab(IN := FALSE);
						sCurrentState.eStep := SP_ManualStp57;
					SP_ManualStp57:
						IF eRobotXYTStatus = AS_InPosition THEN
							TSensorZWaitStab(IN := TRUE, PT := TSensorZWaitStabTime);
							IF TSensorZWaitStab.Q THEN
								IF TSensorMeasure.bInputOutOfRange THEN
									iManMoveAxis:=iManMoveAxisNone;
									sCurrentState.eStep := SP_ManualStp1;
									bZSensorOutOfRangeError := TRUE;
								END_IF
								lrZSensorPosition[iZSensorPositionScan] := TSensorMeasure.lrValue;
								IF iZSensorPositionScan = 0 AND (sPartDataMMI.alrSensorZOffset[1].lrX<>0 OR sPartDataMMI.alrSensorZOffset[1].lrY<>0) THEN
									iZSensorPositionScan := iZSensorPositionScan + 1;
									sCurrentState.eStep := SP_ManualStp56;
								ELSE
									sCurrentState.eStep := SP_ManualStp58;
								END_IF
							END_IF
						END_IF
					SP_ManualStp58: (* Move to take position *)
						IF iZSensorPositionScan = 1 THEN
							(* We used two position, mean the value *)
							ZPositionTakeGive := (lrZSensorPosition[0] + lrZSensorPosition[1]) / 2;
						ELSE
							(* Only one position, use the first one then *)
							ZPositionTakeGive := lrZSensorPosition[0];
						END_IF
						ZPositionTakeGive := alrRobotPos[LTA_Z,LTP_TableSideALayering1] + alrRobotOffset[LTA_Z, iHead] + (lrCalibrationPartAndHeadHeight - sPartDataMMI.lrPartAndHeadHeight) - ZPositionTakeGive;
						alrTargetPos[LA_X] := alrRobotPos[LTA_X,LTP_Lift2] + alrRobotOffset[LTA_X, iHead] + alrLiftCalibrationOffset[LTP_Lift2,LTA_X]  -  sPlateData.alrPartOnPlate[iPlatePos].lrX;
						alrTargetPos[LA_Y] :=alrRobotPos[LTA_Y,LTP_Lift2] + alrRobotOffset[LTA_Y, iHead] + alrLiftCalibrationOffset[LTP_Lift2,LTA_Y] - sPlateData.alrPartOnPlate[iPlatePos].lrY;
						alrTargetPos[LA_THETA] := alrRobotPos[LTA_THETA,LTP_TableSideALayering1] + alrRobotOffset[LTA_THETA, iHead];
						aeMoveRobotCommand[LA_THETA] := AC_MoveAtAbsPos;
						aeMoveRobotCommand[LA_X] := AC_MoveAtAbsPos;
						aeMoveRobotCommand[LA_Y] := AC_MoveAtAbsPos;
						sCurrentState.eStep := SP_ManualStp59;
					SP_ManualStp59:
						IF eRobotXYTStatus = AS_InPosition THEN
							ZPosition := ZPositionTakeGive + sPartDataMMI.lrPartOffsetZLiftDrop;
							sCurrentState.eStep := SP_ManualStp60;
						END_IF
					SP_ManualStp60 : (*Give Part*)
						alrTargetPos[LA_Z1+iHead] := ZPosition + 1;
						aeMoveRobotCommand[LA_Z1+iHead] := AC_MoveAtAbsPos;
						sCurrentState.eStep := SP_ManualStp61;
					SP_ManualStp61 :  (*Movement done*)
						IF aTRobotAxis[LA_Z1+iHead].eCurrentState = AS_InPosition THEN
							 TManualCmd.THead1Vacuum.Activate := FALSE;
							sCurrentState.eStep := SP_ManualStp62;
						END_IF
					SP_ManualStp62:
						(* Check if laying vacuum is disabled *)
						IF aTHeadVacuum[iHead].bVacuumCorrect THEN
							alrTargetPos[LA_Z1+iHead] := alrSafePos[LA_Z1+iHead];
							aeMoveRobotCommand[LA_Z1+iHead] := AC_MoveAtAbsPos;
							sCurrentState.eStep := SP_ManualStp63;
						END_IF
					SP_ManualStp63 :
						IF aTRobotAxis[LA_Z1+iHead].eCurrentState = AS_InPosition THEN
							alrTargetPos[LA_X] := alrRobotPos[LTA_X,LTP_Lift2] + alrRobotOffset[LTA_X, LTO_Vision] + alrLiftCalibrationOffset[LTP_Lift2,LTA_X]  - sPlateData.alrPartOnPlate[iPlatePos].lrX ;
							alrTargetPos[LA_Y] :=  alrRobotPos[LTA_Y,LTP_Lift2] + alrRobotOffset[LTA_Y, LTO_Vision] + alrLiftCalibrationOffset[LTP_Lift2,LTA_Y] - sPlateData.alrPartOnPlate[iPlatePos].lrY ;
							aeMoveRobotCommand[LA_X] := AC_MoveAtAbsPos;
							aeMoveRobotCommand[LA_Y] := AC_MoveAtAbsPos;
							sCurrentState.eStep := SP_ManualStp64;
						END_IF
					SP_ManualStp64:
						IF eRobotXYTStatus = AS_InPosition THEN
							iManMoveAxis:=iManMoveAxisNone;
							sCurrentState.eStep := SP_ManualStp1;
						END_IF
					SP_ManualStp70: (* Move X/Y *)
						aeMoveRobotCommand[LA_X] := AC_MoveAtAbsPos;
						aeMoveRobotCommand[LA_Y] := AC_MoveAtAbsPos;
						sCurrentState.eStep := SP_ManualStp71;
					SP_ManualStp71:
						IF aTRobotAxis[LA_X].eCurrentState= AS_InPosition AND aTRobotAxis[LA_Y].eCurrentState = AS_InPosition THEN
							iManMoveAxis:=iManMoveAxisNone;
							sCurrentState.eStep := SP_ManualStp1;
						END_IF
				END_CASE
				abEnableHeadVacuum[0] := TManualCmd.THead1Vacuum.Activate;
				abEnableHeadVacuum[1] := TManualCmd.THead2Vacuum.Activate;
				bMovePlateTakerDown := TManualCmd.TMovePlateTakerDown.Activate;
				bEnablePlateVacuum := TManualCmd.TPlateVacuum.Activate;
				TManualCmd.lrSensorAdjust := lrSensorAdjust;
				bAspirationBrushOn := TManualCmd.TAspirationBrush.Activate;
			MS_Paused:
				IF bStopReq THEN
					sCurrentState.eStatus := MS_Ready;
				END_IF
		END_CASE;
	MC_Init :
		sCurrentState.eStep := SP_InitStp1;
		sCurrentState.eStatus := MS_Init;
	MC_Run :
		sCurrentState.eStatus := MS_Running;
	MC_Manual :
		sCurrentState.bInitDone := FALSE;
		sCurrentState.eStatus := MS_Manual;
		sCurrentState.eStep := SP_ManualStp0;
	MC_Stop :
		sCurrentState.eStatus := MS_Stopped;
END_CASE;

IF bResetErrors THEN
	sCurrentState.bInError := FALSE;
	bZSensorOutOfRangeError := FALSE;
END_IF

IF bNewJob THEN
	IF C_PROD_MODE_GOOD_PART THEN
		IF sProdLot.dGoodQty > 0 THEN
			sProdLot.dEstimatedPartTime := TIME_TO_DWORD(TJobElapsed)  / sProdLot.dGoodQty;
		ELSE
			sProdLot.dEstimatedPartTime := 0;
		END_IF
	ELSE
		IF sProdLot.dProdQty > 0 THEN
			sProdLot.dEstimatedPartTime := TIME_TO_DWORD(TJobElapsed)  / sProdLot.dProdQty;
		ELSE
			sProdLot.dEstimatedPartTime := 0;
		END_IF
	END_IF
	sProdLot.dLoadedQty := sProdLot.dProdQty;
END_IF

IF bNewJob THEN
(*IF bNewJob OR sCurrentState.eStatus = MS_Manual THEN*)
	abResetPlateState[LPP_Lift1] := TRUE;
	abResetPlateState[LPP_Lift2] := TRUE;
	abResetPlateState[LPP_Reject] := TRUE;
END_IF
IF bNewPlateLift1 THEN abResetPlateState[LPP_Lift1] := TRUE; END_IF
IF bNewPlateLift2 THEN abResetPlateState[LPP_Lift2] := TRUE; END_IF
IF bNewPlateReject THEN abResetPlateState[LPP_Reject] := TRUE; END_IF

IF abCopySwitchFromPlate THEN
	abCopySwitchFromPlate := FALSE;
	FOR j := 0 TO sPlateData.iNbPartOnPlate DO
		aTPartOnSwitchPlate[j].ePartStatus := aTPartOnPlate[LPP_Lift1, j].ePartStatus;
	END_FOR
END_IF

FOR i :=LPP_Reject  TO LPP_Lift2 DO
	IF abResetPlateState[i] THEN
		abResetPlateState[i] := FALSE;
		FOR j := 0 TO sPlateData.iNbPartOnPlate DO
			aTPartOnPlate[i, j ].ePartStatus := PPS_Undefined;
		END_FOR
	END_IF
END_FOR

IF abCopySwitchToPlate THEN
	abCopySwitchToPlate := FALSE;
	FOR j := 0 TO sPlateData.iNbPartOnPlate DO
		aTPartOnPlate[LPP_Lift2, j].ePartStatus := aTPartOnSwitchPlate[j].ePartStatus;
	END_FOR
END_IF
(* ----------------------------------------------------------- MOVE SECURITY CHECK -------------------------------------------------------------------------*)

(* Check if a consequent move more then 2 mm with heads down or plate taker down is requested *)
IF ((ABS(aTRobotAxis[LA_X].lrCurrentPos - alrTargetPos[LA_X]) > lrMaxXYMoveAllowed) AND (aeMoveRobotCommand[LA_X] <> AC_None)) OR
		((ABS(aTRobotAxis[LA_Y].lrCurrentPos - alrTargetPos[LA_Y]) > lrMaxXYMoveAllowed) AND (aeMoveRobotCommand[LA_Y] <> AC_None)) THEN
	IF (aTRobotAxis[LA_Z1].lrCurrentPos > (alrSecuredSafeZPos[0] + lrSafeTolerance))
			OR (aTRobotAxis[LA_Z2].lrCurrentPos > (alrSecuredSafeZPos[1] + lrSafeTolerance))
			OR NOT bPlateTakerIsUp THEN
		IF sCurrentState.eStep <> SP_RunStp63 THEN (* Do not check during cleaning *)
			aeMoveRobotCommand[LA_X] := AC_ForceStop;
			aeMoveRobotCommand[LA_Y] := AC_ForceStop;
			aeMoveRobotCommand[LA_Z1] := AC_ForceStop;
			aeMoveRobotCommand[LA_Z2] := AC_ForceStop;
			sCurrentState.bInitDone := FALSE;
			bConflictDetected := TRUE;
		END_IF
	END_IF
ELSIF ((aTRobotAxis[LA_X].lrCurrentPos > alrUnsecuredArea[0,LA_X]+ lrSafeTolerance) AND (aTRobotAxis[LA_X].lrCurrentPos < alrUnsecuredArea[1,LA_X] - lrSafeTolerance)		(* The Restritcted aera is lrSafeTolerance smaller for the axis have some space to work *)
		AND (aTRobotAxis[LA_Y].lrCurrentPos > alrUnsecuredArea[0,LA_Y]+ lrSafeTolerance) AND (aTRobotAxis[LA_Y].lrCurrentPos < alrUnsecuredArea[1,LA_Y] - lrSafeTolerance)
		AND ((aTRobotAxis[LA_Z1].lrCurrentPos > (alrSafePos[LA_Z1] + lrSafeTolerance))
		OR (aTRobotAxis[LA_Z2].lrCurrentPos > (alrSafePos[LA_Z2] + lrSafeTolerance)))) THEN
	IF (sCurrentState.eStatus = MS_Manual) OR (sCurrentState.eStatus = MS_Init) OR (sCurrentState.eStatus = MS_Stopped) THEN
		bConflictDetected := false;
	ELSE
		aeMoveRobotCommand[LA_X] := AC_ForceStop;
		aeMoveRobotCommand[LA_Y] := AC_ForceStop;
		aeMoveRobotCommand[LA_Z1] := AC_ForceStop;
		aeMoveRobotCommand[LA_Z2] := AC_ForceStop;
		sCurrentState.bInitDone := FALSE;
		bUnsecuredAeraEntry := TRUE;
		bConflictDetected := TRUE;	
	END_IF
END_IF

(* ------------------------------------------------------ END OF MOVE SECURITY CHECK -------------------------------------------------------------------*)

(* Robot command *)

IF (sCurrentState.eStatus = MS_Manual) THEN
	FOR iAxis:=0 TO 4 DO
		IF bManualZIsSafe THEN
			alrRobotSpeed[iAxis] := aTRobotAxis[iAxis].lrFastManualSpeed;
		ELSE
			alrRobotSpeed[iAxis] := aTRobotAxis[iAxis].lrManualSpeed;;
		END_IF
	END_FOR
END_IF

aTRobotAxis[LA_X](
	eCommand 		:= aeMoveRobotCommand[LA_X],
	lrTargetPos 		:= alrTargetPos[LA_X],
	lrTargetSpeed 	:= alrRobotSpeed[LA_X],
	lrAcceleration  := alrRobotAcceleration[LA_X],
	lrDeceleration	:= alrRobotDeceleration[LA_X],
	lrJerk			:= alrRobotJerk[LA_X],
	sAxis		 	:= sXAxisRef,
	bHomeSensor 	:= bHomeX,
	eAxisType		:= AT_AX5000,
	bPowerIsOn		:= bPowerOn,
	bPosLimitSwitch	:= NOT bLimitPosX,
	bNegLimitSwitch	:= NOT bLimitNegX,
	lrMoveOutDist	:= 100,
	bResetErrors	 	:= bResetErrors,
	stServoButton 	:= TManualCmd.aTAxis[LA_X].ServoON
	);
aeMoveRobotCommand[LA_X] := AC_None;
bXAxisError := (aTRobotAxis[LA_X].eCurrentState = AS_InError);

aTRobotAxis[LA_Y](
	eCommand 		:= aeMoveRobotCommand[LA_Y],
	lrTargetPos 		:= alrTargetPos[LA_Y],
	lrTargetSpeed 	:= alrRobotSpeed[LA_Y],
	lrAcceleration  := alrRobotAcceleration[LA_Y],
	lrDeceleration	:= alrRobotDeceleration[LA_Y],
	lrJerk			:= alrRobotJerk[LA_Y],
	sAxis		 	:= sYAxisRef,
	bHomeSensor 	:= bHomeY,
	eAxisType		:= AT_AX5000,
	bPowerIsOn		:= bPowerOn,
	bPosLimitSwitch	:= NOT bLimitPosY,
	bNegLimitSwitch	:= NOT bLimitNegY,
	lrMoveOutDist	:= 100,
	bResetErrors	 	:= bResetErrors,
	stServoButton 	:= TManualCmd.aTAxis[LA_Y].ServoON

);
aeMoveRobotCommand[LA_Y] := AC_None;
bYAxisError := (aTRobotAxis[LA_Y].eCurrentState = AS_InError);

aTRobotAxis[LA_Z1](
	eCommand 		:= aeMoveRobotCommand[LA_Z1],
	lrTargetPos 		:= alrTargetPos[LA_Z1],
	lrTargetSpeed 	:= alrRobotSpeed[LA_Z1],
	sAxis	 		:= sZ1AxisRef,
	bHomeSensor 	:= bHomeZ1,
	bPowerIsOn		:= bPowerOn,
	bPosLimitSwitch	:= NOT bLimitPosZ1,
	bNegLimitSwitch	:= NOT bLimitNegZ1,
	lrMoveOutDist	:= 10,
	bResetErrors	 	:= bResetErrors,
	stServoButton 	:= TManualCmd.aTAxis[LA_Z1].ServoON
);
aeMoveRobotCommand[LA_Z1] := AC_None;
bZ1AxisError := (aTRobotAxis[LA_Z1].eCurrentState = AS_InError);

aTRobotAxis[LA_Z2](
	eCommand 		:= aeMoveRobotCommand[LA_Z2],
	lrTargetPos 		:= alrTargetPos[LA_Z2],
	lrTargetSpeed 	:= alrRobotSpeed[LA_Z2],
	sAxis		 	:= sZ2AxisRef,
	bHomeSensor 	:= bHomeZ2,
	bPowerIsOn		:= bPowerOn,
	bPosLimitSwitch	:= NOT bLimitPosZ2,
	bNegLimitSwitch	:= NOT bLimitNegZ2,
	lrMoveOutDist	:= 10,
	bResetErrors	 	:= bResetErrors,
	stServoButton 	:= TManualCmd.aTAxis[LA_Z2].ServoON
);
aeMoveRobotCommand[LA_Z2] := AC_None;
bZ2AxisError := (aTRobotAxis[LA_Z2].eCurrentState = AS_InError);

aTRobotAxis[LA_THETA](
	eCommand 		:= aeMoveRobotCommand[LA_THETA],
	lrTargetPos 		:= alrTargetPos[LA_THETA],
	lrTargetSpeed 	:= alrRobotSpeed[LA_THETA],
	sAxis		 	:= sThetaAxisRef,
	bPowerIsOn		:= bPowerOn,
	bResetErrors	 	:= bResetErrors,
	eHomingAxisType := AHT_OnZeroEncoder,
	stServoButton 	:= TManualCmd.aTAxis[LA_THETA].ServoON
);
aeMoveRobotCommand[LA_THETA] := AC_None;
bTAxisError := (aTRobotAxis[LA_THETA].eCurrentState = AS_InError);

(* Get move result *)
eRobotXYTStatus := AS_Moving;
IF (aTRobotAxis[LA_X].eCurrentState = AS_InError) OR (aTRobotAxis[LA_Y].eCurrentState = AS_InError) OR (aTRobotAxis[LA_THETA].eCurrentState = AS_InError) THEN
	eRobotXYTStatus := AS_InError;
ELSIF (aTRobotAxis[LA_X].eCurrentState = AS_InPosition) AND (aTRobotAxis[LA_Y].eCurrentState = AS_InPosition) AND (aTRobotAxis[LA_THETA].eCurrentState = AS_InPosition) THEN
		eRobotXYTStatus := AS_InPosition;
END_IF

(* Handle part vacuum *)
aTHeadVacuum[0](
	bEnableVacuum		:= abEnableHeadVacuum[0],
	tVacErrorDelay		:= INT_TO_TIME(sVaccumSettingsHead.iErrorDelay),
	tBlowingTime			:= INT_TO_TIME(sVaccumSettingsHead.iBlowing),
	tWaitVacuumOK		:= INT_TO_TIME(sVaccumSettingsHead.iWaitWhenVacuumOk),
	bReset				:= bResetErrors  OR abResetVacuum[0],
	iVacuum				:= iHead1VacuumFlow,
	lrVacuumThreshold	 :=  alrVacuumThreshold[0],
	bDisableVacuumChecking := abBypassVacuumError[0],
	bVacuumOn			=> bActivateHead1Vacuum,
	bBlowOn				=> bActivateHead1Blowing,
	bVacuumError		=> bHead1VacuumError
);
abResetVacuum[0] := FALSE;
IF abBypassVacuumError[0] AND sCurrentState.eStatus = MS_Running THEN
	bHead1VacuumError := FALSE;
END_IF
IF (bResetErrors AND (sCurrentState.eStatus = MS_Stopped) AND bHead1VacuumError) THEN
	abEnableHeadVacuum[0] := FALSE;
END_IF

aTHeadVacuum[1](
	bEnableVacuum		:= abEnableHeadVacuum[1],
	tVacErrorDelay		:= INT_TO_TIME(sVaccumSettingsHead.iErrorDelay),
	tBlowingTime			:= INT_TO_TIME(sVaccumSettingsHead.iBlowing),
	tWaitVacuumOK		:= INT_TO_TIME(sVaccumSettingsHead.iWaitWhenVacuumOk),
	bReset				:= bResetErrors  OR abResetVacuum[1],
	iVacuum				:= iHead2VacuumFlow,
	lrVacuumThreshold	 :=  alrVacuumThreshold[1],
	bDisableVacuumChecking := abBypassVacuumError[1],
	bVacuumOn			=> bActivateHead2Vacuum,
	bBlowOn				=> bActivateHead2Blowing,
	bVacuumError		=> bHead2VacuumError
);
abResetVacuum[1] := FALSE;
IF abBypassVacuumError[1] AND sCurrentState.eStatus = MS_Running THEN
	bHead2VacuumError := FALSE;
END_IF
IF (bResetErrors AND (sCurrentState.eStatus = MS_Stopped) AND bHead2VacuumError) THEN
	abEnableHeadVacuum[1] := FALSE;
END_IF

(* Handle plate vacuum *)
TPlateVacuum(
	tVacErrorDelay		:= INT_TO_TIME(sVaccumSettingsPlate.iErrorDelay),
	tBlowingTime			:= INT_TO_TIME(sVaccumSettingsPlate.iBlowing),
	tWaitVacuumOK		:= INT_TO_TIME(sVaccumSettingsPlate.iWaitWhenVacuumOk),
	bEnableVacuum	:= bEnablePlateVacuum,
	bReset			:= bResetErrors,
	bVacuumOK		:= bPlateVacuumIsOk,
	bVacuumOn		=> bActivatePlateVacuum,
	bBlowOn			=> bActivatePlateBlowing,
	bVacuumError	=> bPlateVacuumError
);

(* Check jack error *)
TCheckJack(
	bJackGoOut	:= bMovePlateTakerDown,
	bJackIsIn	:= bPlateTakerIsUp,
	bJackIsOut	:= bPlateTakerIsDown,
	tTimeOut		:= t#2s,
	bResetErrors := bResetErrors,
	bJackError	=> bJackError
);

IF bJackError OR bXAxisError OR bYAxisError OR bZ1AxisError OR bZ2AxisError OR bTAxisError OR bHead1VacuumError OR bHead2VacuumError OR bPlateVacuumError OR bConflictDetected  OR bZSensorOutOfRangeError THEN
	sCurrentState.bInError := TRUE;
	IF (sCurrentState.eStatus <> MS_Manual) AND (sCurrentState.eStatus <> MS_Stopped) AND (sCurrentState.eStatus <> MS_Init) THEN
		sCurrentState.eStatus := MS_Ready;
	END_IF
END_IF

IF (NOT bPowerOn OR bXAxisError OR bYAxisError OR bZ1AxisError OR bZ2AxisError OR bTAxisError) THEN
	sCurrentState.bInitDone := FALSE;
	IF (sCurrentState.eStatus <> MS_Manual) THEN
		sCurrentState.eStatus := MS_Stopped;
	END_IF
END_IF

IF bNewJob THEN
(*	sProdLot.dProdQty := 0;
	sProdLot.dGoodQty := 0;
	sProdLot.dLoadedQty := 0; *)
	sProdLot.dEstimatedTimeLeft := 0;
END_IF
sProdLot.dProductionTime := TIME_TO_DWORD(TJobElapsed);

CASE sRunData.eModule OF
	LMP_Table:
		sOutGiveToTable := sOutGiveToModule;
		sOutTakeFromTable := sOutTakeFromModule;
	LMP_TurnOverFix,LMP_TurnOverArm:
		sOutGiveToTurnOver := sOutGiveToModule;
		sOutTakeFromTurnOver := sOutTakeFromModule;
END_CASE

(* Detect if lift seems to move to refresh Z position *)
IF eLift1RunStatus <> RS_WaitRequest THEN
	alrZLiftPos[LTP_Lift1] := 0;
END_IF
IF eLift2RunStatus <> RS_WaitRequest THEN
	alrZLiftPos[LTP_Lift2] := 0;
END_IF

sRunData.lrZPositionTakeGive := ZPositionTakeGive;
bVacuumInUse := bEnablePlateVacuum OR (abEnableHeadVacuum[0] AND NOT bHead1VacuumError)  OR (abEnableHeadVacuum[1] AND NOT bHead2VacuumError) ;
bMovePlateTakerUp := NOT bMovePlateTakerDown;

sCurrentState.bInterlocked := bManInterlock AND  (sCurrentState.eStatus = MS_Manual);
bModuleError := sCurrentState.bInError;
sCurrentState.bRunning := (sCurrentState.eStatus = MS_Running);
IF (sCurrentState.eStatus <> MS_Running) THEN eRunStatus := RS_NotRunning; END_IF

iStep := sCurrentState.eStep;

END_FUNCTION_BLOCK

// ---- POUs/Drivers/StdAxis.TcPOU
FUNCTION_BLOCK StdAxis

(*
	Description 	: Bloc fonction de gestion d'un axe
	Auteur		: DRE
	Date		: 30.08.2016
	Version		: 1.00

	Modifications :

*)

VAR_INPUT
	eCommand				: TAxisCommands;					(* Commande d'axe à exécuter *)
	lrTargetPos				: LREAL;								(* Position cible *)
	lrTargetSpeed			: LREAL;								(* Vitesse cible *)
	lrAcceleration 			: LREAL		:= 0;						(* Accélération pour le nouveau mouvement *)
	lrDeceleration 			: LREAL		:= 0;						(* Décélération pour le nouveau mouvement *)
	lrJerk 					: LREAL		:= 0;						(* Facteur saccade pour le nouveau mouvement *)
	bResetErrors				: BOOL;								(* MAZ de l'erreur générale du bloc *)
	bHomeSensor			: BOOL;								(* Capteur de home *)
	bPowerIsOn				: BOOL;									(* Alimentation principale présente *)
	eAxisType				: TAxisType	:= AT_Standard;			(* Type d'axe *)
	eHomingAxisType		: TAxisHomingType := AHT_OnSensor;	(*Type de homing *)
	bPosLimitSwitch			: BOOL		:= FALSE;				(* Limit switch côté positif actif *)
	bNegLimitSwitch			: BOOL		:= FALSE;				(* Limit switch côté negatif actif *)
	lrMoveOutDist			: LREAL		:= 0;						(* Distance to move out when on switch *)
	bResetUseTime			: BOOL		:= FALSE;
END_VAR
VAR_OUTPUT
	eCurrentState				: TAxisState	:= AS_PowerOff;
	lrCurrentPos				: LREAL;
	lrMinPos					: LREAL;
	bMinPosMonitoring		: BOOL;
	lrMaxPos				: LREAL;
	bMaxPosMonitoring		: BOOL;
	lrManualSpeed			: LREAL;
	lrFastManualSpeed		: LREAL;
	lrRunningSpeed			: LREAL;
	lrRemainingTimeToGo		: LREAL;
	dwUseHours				: DWORD;
END_VAR
VAR_IN_OUT
	sAxis					: AXIS_REF;							(* Bloc de données entre NC et PLC*)
	stServoButton				: TManButton;
END_VAR
VAR
	bServoOn				: BOOL;
	bHome					: BOOL;
	bMoveVel				: BOOL;
	bMoveAbs				: BOOL;
	bMoveRel				: BOOL;
	bMoveModulo			: BOOL;
	bStop					: BOOL;
	bHalt					: BOOL;
	bSetPosition				: BOOL;
	bAxisReady				: BOOL;
	bAxisHomed				: BOOL;
	bRemoveLimitSecurity		: BOOL;
	i						: INT;
	iUseBlock				: INT;
	afbMoveAbs				: ARRAY[0..1] OF MC_MoveAbsolute;
	afbMoveModulo			: ARRAY[0..1] OF MC_MoveModulo;
	afbMoveRel				: ARRAY[0..1] OF MC_MoveRelative;
	afbMoveVel				: ARRAY[0..1] OF MC_MoveVelocity;
	afbStop					: ARRAY[0..1] OF MC_Stop;
	afbHalt					: ARRAY[0..1] OF MC_Halt;
	fbPower					: MC_PowerStepper;
	fbReadPos				: MC_ReadActualPosition;
	fbReset					: MC_Reset;
	fbHome					: MC_Home;
	fbResetSOE				: FB_SoEReset;
	fbSetPosition				: MC_SetPosition;
	fbReadParamTimeToGo	: MC_ReadParameter;
(*	fbReadParamModulo		: MC_ReadParameter;
	fbReadParamMinPos		: MC_ReadParameter;
	fbReadParamMaxPos		: MC_ReadParameter; *)
	fbReadParameters		: MC_ReadParameterSet;
	fbReadStatus				: MC_ReadStatus;
	lrPosition					: LREAL;
	lrSpeed					: LREAL := 100;
	lrModuloValue			: LREAL;
	eMoveDir				: MC_Direction;
	TCheckReady			: TON;
	eLastCurrentState			: TAxisState	:= AS_PowerOff;
	eInitCommand			: TAxisCommands;					(* Commande d'axe à exécuter lors du homing *)
	lrInitTargetPos			: LREAL;
	lrInitTargetSpeed			: LREAL;
	lrLimitOutSpeed			: LREAL;						(* Speed to move out of limit switch *)
	eHomingMode			: MC_HomingMode := MC_DefaultHoming;
	ePowerCommand			: TAxisCommands;
	stReadAxisParameters		: ST_AxisParameterSet;
	stAxisParameters			: ST_AxisParameterSet;
	eStep					: TModuleSteps := SP_RunStp0;
	bFirstCycleState			: BOOL;
	bReadParameters		: BOOL;
	bReadParametersOnce	: BOOL; (*Make sure we have read the parameters at least one before moving or homing *)
	iStep					: INT;
	iState					: INT;
	lrHomingSearchMin		: LREAL;
	lrHomingSearchMax		: LREAL;
	lrHomingOffset			: LREAL;
	lrHomingPercent			: LREAL;
	lrUnitMotorTurn			: LREAL;
	bSearchHoming			: BOOL;
	bMoveLimitNeg			: BOOL;
	bMoveToLimitNegRequest	: BOOL;
	lrCurrentMovingSpeed		: LREAL;
	iDebugPos				: INT;
	TUseCounter				: RunningCounter;
END_VAR

(* Some  FB that can be usefull
MC_Jog
MC_ReadStatus
*)

TUseCounter(bStart := bServoOn, bReset := bResetUseTime);
dwUseHours := TUseCounter.dwHours;

IF (bSearchHoming) THEN
	eCommand := AC_MoveHome;
	bSearchHoming := FALSE;
END_IF
IF (bMoveLimitNeg) THEN
	eCommand := AC_MoveLimitNeg;
	bMoveLimitNeg := FALSE;
END_IF

IF eCommand =AC_ClearPosition THEN
	bSetPosition := TRUE;
	lrPosition := 0;
END_IF

(* Manual Handling*)
IF eCommand = AC_None THEN
	IF stServoButton.Activate AND eCurrentState = AS_PowerOff AND eCurrentState = eLastCurrentState THEN
		eCommand := AC_ServoOn;
	ELSIF NOT stServoButton.Activate AND ((eCurrentState = AS_Powering  AND eCurrentState = eLastCurrentState) OR eCurrentState = AS_NotHomed OR eCurrentState = AS_InPosition OR eCurrentState = AS_OnLimitNeg) THEN
		eCommand := AC_ServoOff;
	END_IF
END_IF

(*check external command during homing *)
IF eCurrentState = AS_Homing OR eCurrentState = AS_MovingHoming OR eCurrentState = AS_MovingLimitNeg THEN
	CASE eCommand OF
		AC_ForceStop, AC_ServoOff:
			eInitCommand := eCommand;
		AC_MoveLimitNeg:
			IF eCurrentState = AS_Homing THEN
				bMoveToLimitNegRequest := TRUE;
			END_IF
	END_CASE
	eCommand := eInitCommand ; (*Use internal command during homing*)
	eInitCommand := AC_None;
	lrTargetPos := lrInitTargetPos;
	lrTargetSpeed := lrInitTargetSpeed;
END_IF

(*Handle move command *)
IF eCurrentState = AS_InPosition OR eCurrentState = AS_Moving OR  eCurrentState = AS_Homing OR eCurrentState = AS_MovingHoming OR eCurrentState = AS_MovingLimitNeg THEN
	CASE eCommand OF
		AC_MoveAtSpeed:
			iUseBlock := (iUseBlock + 1) MOD 2;
			bMoveVel 		:= TRUE;
			bMoveAbs 		:= FALSE;
			bMoveRel 		:= FALSE;
			bMoveModulo 	:= FALSE;
			bStop 			:= FALSE;
			bHalt			:= FALSE;
			lrPosition := lrTargetPos;
			lrSpeed := lrTargetSpeed;
			lrCurrentMovingSpeed := lrSpeed;
			IF (lrPosition < 0) THEN
				eMoveDir := MC_Negative_Direction;
			ELSE
				eMoveDir := MC_Positive_Direction;
			END_IF
		AC_MoveAtRelPos:
			iUseBlock := (iUseBlock + 1) MOD 2;
			bMoveVel 		:= FALSE;
			bMoveAbs 		:= FALSE;
			bMoveRel 		:= TRUE;
			bMoveModulo 	:= FALSE;
			bStop 			:= FALSE;
			bHalt			:= FALSE;
			lrPosition := lrTargetPos;
			lrSpeed := lrTargetSpeed;
			lrCurrentMovingSpeed := lrSpeed;
		AC_MoveAtAbsPos:
			iUseBlock := (iUseBlock + 1) MOD 2;
			bMoveVel 		:= FALSE;
			bMoveAbs 		:= TRUE;
			bMoveRel 		:= FALSE;
			bMoveModulo 	:= FALSE;
			bStop 			:= FALSE;
			bHalt			:= FALSE;
			lrPosition := lrTargetPos;
			lrSpeed := lrTargetSpeed;
			lrCurrentMovingSpeed := lrSpeed;
		AC_MoveModulo:
			iUseBlock := (iUseBlock + 1) MOD 2;
			bMoveVel 		:= FALSE;
			bMoveAbs 		:= FALSE;
			bMoveRel 		:= FALSE;
			bMoveModulo 	:= TRUE;
			bStop 			:= FALSE;
			bHalt			:= FALSE;
			lrPosition := lrTargetPos;
			lrSpeed := lrTargetSpeed;
			lrCurrentMovingSpeed := lrSpeed;
			IF (lrPosition < 0) THEN
	 			lrPosition := LMOD(lrPosition,lrModuloValue) + lrModuloValue;
			END_IF
			IF (lrPosition >= lrModuloValue) THEN
				lrPosition := LMOD(lrPosition,lrModuloValue);
			END_IF
		AC_Stop:
			iUseBlock := (iUseBlock + 1) MOD 2;
			bMoveVel 		:= FALSE;
			bMoveAbs 		:= FALSE;
			bMoveRel 		:= FALSE;
			bMoveModulo 	:= FALSE;
			bStop 			:= FALSE;
			bHalt			:= TRUE;
			lrCurrentMovingSpeed := lrSpeed;
		AC_ForceStop:
			eCurrentState := AS_Stopping;
	END_CASE
END_IF

IF (eCurrentState <> eLastCurrentState) THEN
	eStep := SP_RunStp0;
	eLastCurrentState := eCurrentState;
	bFirstCycleState := TRUE;
ELSE
	bFirstCycleState := FALSE;
END_IF

CASE eCurrentState OF
	AS_PowerOff:
		bRemoveLimitSecurity := FALSE;
		bServoOn 		:= FALSE;
		bHome			:= FALSE;
		bMoveVel 		:= FALSE;
		bMoveAbs 		:= FALSE;
		bMoveRel 		:= FALSE;
		bMoveModulo 	:= FALSE;
		bStop 			:= FALSE;
		bHalt			:= FALSE;
		bSetPosition 		:= FALSE;
		IF ePowerCommand = AC_Init OR ePowerCommand = AC_MoveLimitNeg THEN (* continue if we have receive an init command during the reseting step *)
			eCommand := ePowerCommand;
		END_IF
		CASE eCommand OF
			AC_ServoOn, AC_Init, AC_MoveLimitNeg:
				ePowerCommand := eCommand;
				eCurrentState := AS_Powering;
		END_CASE
	AS_Powering:
		IF eCommand = AC_Init OR eCommand = AC_MoveLimitNeg THEN
			ePowerCommand := eCommand;
		END_IF
		CASE eStep OF
			SP_RunStp0:
				bServoOn := TRUE;
				bRemoveLimitSecurity := bPosLimitSwitch OR bNegLimitSwitch;
				TCheckReady(IN := FALSE);
				eStep := SP_RunStp1;
			SP_RunStp1:
				TCheckReady(IN := TRUE, PT := t#10s);
				IF TCheckReady.Q THEN
					eCurrentState := AS_InError;
					iDebugPos := 1;
				ELSIF bAxisReady AND bReadParametersOnce THEN
					CASE ePowerCommand OF (*Check what command trig the power on *)
						AC_ServoOn:
							IF bAxisHomed THEN
								eCurrentState := AS_InPosition;
							ELSE
								eCurrentState := AS_NotHomed;
							END_IF
						AC_Init:
							IF bAxisHomed THEN
								eCurrentState := AS_InPosition;
							ELSE
								eCurrentState := AS_Homing;
							END_IF
						AC_MoveLimitNeg:
							eCurrentState := AS_MovingLimitNeg;
					END_CASE
					ePowerCommand := AC_None; (* clear previous command *)
				END_IF
		END_CASE
		IF eCommand = AC_ServoOff THEN
			ePowerCommand := AC_None; (* clear previous command *)
			eCurrentState := AS_PowerOff;
		END_IF
	AS_NotHomed:
		CASE eCommand OF
			AC_ServoOff:
				eCurrentState := AS_PowerOff;
			AC_Init, AC_Home:
				eCurrentState := AS_Homing;
			AC_MoveLimitNeg:
				eCurrentState := AS_MovingLimitNeg;
		END_CASE
		IF NOT bAxisReady THEN
			iDebugPos := 2;
			eCurrentState := AS_InError;
		END_IF
	AS_Homing:
		CASE eStep OF
			SP_RunStp0:
				bHome := FALSE;
				IF eHomingAxisType = AHT_NoHoming THEN
					eStep := SP_RunStp30;
				ELSE
					eStep := SP_RunStp1;
				END_IF
			SP_RunStp1:
				IF lrMoveOutDist = 0 THEN
					eStep := SP_RunStp30;
				ELSIF bPosLimitSwitch THEN
					lrPosition := lrMoveOutDist+1;
					bSetPosition := TRUE;
					eStep := SP_RunStp10;
				ELSIF bNegLimitSwitch THEN
					lrPosition :=  -lrMoveOutDist-1;
					bSetPosition := TRUE;
					eStep := SP_RunStp20;
				ELSE
					eStep := SP_RunStp30;
				END_IF
			SP_RunStp10:
				IF fbSetPosition.Done THEN
					lrInitTargetSpeed := lrLimitOutSpeed;
					lrInitTargetPos := -lrMoveOutDist;
					eInitCommand := AC_MoveAtRelPos;
					eStep := SP_RunStp11;
				END_IF
			SP_RunStp11:
				IF afbMoveRel[iUseBlock].Done THEN
					eStep := SP_RunStp30;
				ELSIF afbMoveRel[iUseBlock].CommandAborted THEN
					iDebugPos := 3;
					eCurrentState := AS_InError;
				END_IF
			SP_RunStp20:
				IF fbSetPosition.Done THEN
					lrInitTargetSpeed := lrLimitOutSpeed;
					lrInitTargetPos := lrMoveOutDist;
					eInitCommand := AC_MoveAtRelPos;
					eStep := SP_RunStp21;
				END_IF
			SP_RunStp21:
				IF afbMoveRel[iUseBlock].Done THEN
					eStep := SP_RunStp30;
				ELSIF afbMoveRel[iUseBlock].CommandAborted THEN
					iDebugPos := 4;
					eCurrentState := AS_InError;
				END_IF
			SP_RunStp30:
				bRemoveLimitSecurity := FALSE;
				bHome := TRUE;
				CASE eHomingAxisType OF
					AHT_NoHoming:
						eHomingMode	:= MC_ForceCalibration;
					AHT_OnSensor:
						eHomingMode	:= MC_DefaultHoming;
					AHT_OnZeroEncoder:
						eHomingMode	:= MC_DefaultHoming;
						bHomeSensor := TRUE;
				END_CASE
				eStep := SP_RunStp31;
			SP_RunStp31:
				IF (eHomingAxisType = AHT_OnZeroEncoder) THEN
					bHomeSensor := NOT (sAxis.NcToPlc.HomingState >= 4);
				END_IF
				IF fbHome.Done THEN
					bHome := FALSE;
					bAxisHomed := TRUE;
					IF bMoveToLimitNegRequest THEN
						eCurrentState := AS_MovingLimitNeg;
						bMoveToLimitNegRequest := FALSE;
					ELSE
						eCurrentState := AS_InPosition;
					END_IF
				END_IF
		END_CASE
		IF NOT bAxisReady THEN
			iDebugPos := 5;
			eCurrentState := AS_InError;
		END_IF
	AS_InPosition:
		CASE eCommand OF
			AC_MoveAtSpeed, AC_MoveAtRelPos, AC_MoveAtAbsPos, AC_MoveModulo, AC_Stop:
				eCurrentState := AS_Moving;
			AC_ServoOff:
				eCurrentState := AS_PowerOff;
			AC_Home:
				eCurrentState := AS_Homing;
			AC_MoveHome:
				IF (eHomingAxisType = AHT_OnSensor) THEN
					eCurrentState := AS_MovingHoming;
				END_IF
			AC_MoveLimitNeg:
				eCurrentState := AS_MovingLimitNeg;
		END_CASE
		IF NOT bAxisReady THEN
			iDebugPos := 6;
			eCurrentState := AS_InError;
		END_IF
	AS_Moving:
		IF eCommand = AC_MoveLimitNeg THEN
			bMoveToLimitNegRequest := TRUE;
		END_IF
		IF NOT ((eCommand = AC_MoveAtSpeed) OR (eCommand = AC_MoveAtRelPos) OR (eCommand = AC_MoveAtAbsPos) OR (eCommand = AC_MoveModulo) OR (eCommand = AC_Stop)) THEN (* Not a move command *)
			FOR i:=0 TO 1 DO
				IF afbMoveAbs[iUseBlock].Done OR afbMoveModulo[iUseBlock].Done OR afbMoveRel[iUseBlock].Done OR afbStop[iUseBlock].Done OR afbHalt[iUseBlock].Done THEN
					bMoveVel 		:= FALSE;
					bMoveAbs 		:= FALSE;
					bMoveRel 		:= FALSE;
					bMoveModulo 	:= FALSE;
					bStop 			:= FALSE;
					bHalt			:= FALSE;
					IF bMoveToLimitNegRequest THEN
						eCurrentState := AS_MovingLimitNeg;
						bMoveToLimitNegRequest := FALSE;
					ELSE
						eCurrentState := AS_InPosition;
					END_IF
				END_IF
			END_FOR
			FOR i:=0 TO 1 DO
				IF afbMoveAbs[iUseBlock].CommandAborted OR afbMoveModulo[iUseBlock].CommandAborted OR afbMoveRel[iUseBlock].CommandAborted OR afbStop[iUseBlock].CommandAborted OR afbHalt[iUseBlock].CommandAborted THEN
					iDebugPos := 7;
					eCurrentState := AS_InError;
				END_IF
			END_FOR
			IF lrCurrentMovingSpeed <> lrTargetSpeed AND eCurrentState = AS_Moving AND ABS(lrTargetPos-lrCurrentPos)>0.1 THEN
				(* switch block to update speed *)
				lrCurrentMovingSpeed := lrTargetSpeed;
				lrSpeed := lrTargetSpeed;
				iUseBlock := (iUseBlock + 1) MOD 2;
			END_IF
			(*IF NOT fbReadStatus.Status.HasJob AND eCurrentState = AS_Moving AND NOT bFirstCycleState THEN
				iDebugPos := 8;
				eCurrentState := AS_InError;
			END_IF*)
		END_IF
		IF NOT bAxisReady THEN
			iDebugPos := 9;
			eCurrentState := AS_InError;
		END_IF
	AS_MovingHoming:
		CASE eStep OF
			SP_RunStp0 :  (* Init Data*)
				lrHomingOffset := 0;
				IF stAxisParameters.nEncMaxIncrement = 16#FFFFFFFF THEN
					lrUnitMotorTurn := stAxisParameters.fEncScaleFactorInternal * DWORD_TO_LREAL(16#000FFFFF+1);
				ELSE
					lrUnitMotorTurn := stAxisParameters.fEncScaleFactorInternal * DWORD_TO_LREAL(stAxisParameters.nEncMaxIncrement+1);
				END_IF

